KUKA KRL program: Kuka_Relative_Mo1.src

&ACCESS RVP
&REL 1
&PARAM TEMPLATE = C:\KRC\Roboter\Template\vorgabe
&PARAM EDITMASK = *
DEF Kuka_Relative_Mo1 ( )

; External program calls:
EXT Kuka_Relative_Mo2()

; $TOOL = TOOL_DATA[1]
; --------------------------
PTP {A1 -96.46360,A2 -64.41550,A3 114.80900,A4 -13.88510,A5 -54.29400,A6 -19.74150}
; ---- Setting reference (Base) ----
$BASE = {FRAME: X 0.000,Y 0.000,Z 0.000,A 0.000,B 0.000,C 0.000}
; --------------------------
; ---- Setting tool (TCP) ----
; TOOL_DATA[1] = {FRAME: X 0.000,Y 0.000,Z 10.000,A 0.000,B 0.000,C 0.000}
$TOOL = {FRAME: X 0.000,Y 0.000,Z 10.000,A 0.000,B 0.000,C 0.000}
; $TOOL = TOOL_DATA[1]
; --------------------------
PTP {A1 -96.46360,A2 -64.41550,A3 114.80900,A4 -13.88510,A5 -54.29400,A6 40.25850}
; ---- Setting reference (Base) ----
$BASE = {FRAME: X 0.000,Y 0.000,Z 0.000,A 0.000,B 0.000,C 0.000}
; --------------------------
; ---- Setting tool (TCP) ----
; TOOL_DATA[1] = {FRAME: X 0.000,Y 0.000,Z 10.000,A 0.000,B 0.000,C 0.000}
$TOOL = {FRAME: X 0.000,Y 0.000,Z 10.000,A 0.000,B 0.000,C 0.000}
; $TOOL = TOOL_DATA[1]
; --------------------------
PTP {A1 -96.46360,A2 -64.41550,A3 114.80900,A4 -13.88510,A5 -54.29400,A6 10.25850}
; ---- Setting reference (Base) ----
$BASE = {FRAME: X 0.000,Y 0.000,Z 0.000,A 0.000,B 0.000,C 0.000}
; --------------------------
; ---- Setting tool (TCP) ----
; TOOL_DATA[1] = {FRAME: X 0.000,Y 0.000,Z 10.000,A 0.000,B 0.000,C 0.000}
$TOOL = {FRAME: X 0.000,Y 0.000,Z 10.000,A 0.000,B 0.000,C 0.000}
; $TOOL = TOOL_DATA[1]
; --------------------------
PTP {A1 -85.55830,A2 -64.18770,A3 116.67500,A4 -0.42100,A5 -55.51980,A6 1.70277}
; ---- Setting reference (Base) ----
$BASE = {FRAME: X 0.000,Y 0.000,Z 0.000,A 0.000,B 0.000,C 0.000}
; --------------------------
; ---- Setting tool (TCP) ----
; TOOL_DATA[1] = {FRAME: X 0.000,Y 0.000,Z 10.000,A 0.000,B 0.000,C 0.000}
$TOOL = {FRAME: X 0.000,Y 0.000,Z 10.000,A 0.000,B 0.000,C 0.000}
; $TOOL = TOOL_DATA[1]
; --------------------------
PTP {A1 -90.55220,A2 -62.64360,A3 114.04900,A4 -40.68250,A5 -62.48120,A6 23.77200}
; ---- Setting reference (Base) ----
$BASE = {FRAME: X 0.000,Y 0.000,Z 0.000,A 0.000,B 0.000,C 0.000}
; --------------------------
; ---- Setting tool (TCP) ----
; TOOL_DATA[1] = {FRAME: X 0.000,Y 0.000,Z 10.000,A 0.000,B 0.000,C 0.000}
$TOOL = {FRAME: X 0.000,Y 0.000,Z 10.000,A 0.000,B 0.000,C 0.000}
; $TOOL = TOOL_DATA[1]
; --------------------------
PTP {A1 -80.54180,A2 -63.03590,A3 114.13400,A4 40.72610,A5 -60.63820,A6 -21.43390}
; ---- Setting reference (Base) ----
$BASE = {FRAME: X 0.000,Y 0.000,Z 0.000,A 0.000,B 0.000,C 0.000}
; --------------------------
; ---- Setting tool (TCP) ----
; TOOL_DATA[1] = {FRAME: X 0.000,Y 0.000,Z 10.000,A 0.000,B 0.000,C 0.000}
$TOOL = {FRAME: X 0.000,Y 0.000,Z 10.000,A 0.000,B 0.000,C 0.000}
; $TOOL = TOOL_DATA[1]
; --------------------------
PTP {A1 -85.55830,A2 -64.18770,A3 116.67500,A4 -0.42100,A5 -55.51980,A6 1.70277}
; ---- Setting reference (Base) ----
$BASE = {FRAME: X 0.000,Y 0.000,Z 0.000,A 0.000,B 0.000,C 0.000}
; --------------------------
; ---- Setting tool (TCP) ----
; TOOL_DATA[1] = {FRAME: X 0.000,Y 0.000,Z 10.000,A 0.000,B 0.000,C 0.000}
$TOOL = {FRAME: X 0.000,Y 0.000,Z 10.000,A 0.000,B 0.000,C 0.000}
; $TOOL = TOOL_DATA[1]
; --------------------------
PTP {A1 -85.55830,A2 -64.18770,A3 116.67500,A4 -0.42100,A5 -55.51980,A6 -28.29720}
; ---- Setting reference (Base) ----
$BASE = {FRAME: X 0.000,Y 0.000,Z 0.000,A 0.000,B 0.000,C 0.000}
; --------------------------
; ---- Setting tool (TCP) ----
; TOOL_DATA[1] = {FRAME: X 0.000,Y 0.000,Z 10.000,A 0.000,B 0.000,C 0.000}
$TOOL = {FRAME: X 0.000,Y 0.000,Z 10.000,A 0.000,B 0.000,C 0.000}
; $TOOL = TOOL_DATA[1]
; --------------------------
PTP {A1 -85.55830,A2 -64.18770,A3 116.67500,A4 -0.42100,A5 -55.51980,A6 31.70280}
; ---- Setting reference (Base) ----
$BASE = {FRAME: X 0.000,Y 0.000,Z 0.000,A 0.000,B 0.000,C 0.000}
; --------------------------
; ---- Setting tool (TCP) ----
; TOOL_DATA[1] = {FRAME: X 0.000,Y 0.000,Z 10.000,A 0.000,B 0.000,C 0.000}
$TOOL = {FRAME: X 0.000,Y 0.000,Z 10.000,A 0.000,B 0.000,C 0.000}
; $TOOL = TOOL_DATA[1]
; --------------------------
PTP {A1 -85.55830,A2 -64.18770,A3 116.67500,A4 -0.42100,A5 -55.51980,A6 1.70277}
; ---- Setting reference (Base) ----
$BASE = {FRAME: X 0.000,Y 0.000,Z 0.000,A 0.000,B 0.000,C 0.000}
; --------------------------
; ---- Setting tool (TCP) ----
; TOOL_DATA[1] = {FRAME: X 0.000,Y 0.000,Z 10.000,A 0.000,B 0.000,C 0.000}
$TOOL = {FRAME: X 0.000,Y 0.000,Z 10.000,A 0.000,B 0.000,C 0.000}
; $TOOL = TOOL_DATA[1]
; --------------------------
PTP {A1 -86.78140,A2 -64.12760,A3 116.64400,A4 -1.90174,A5 -55.56400,A6 2.60482}
; ---- Setting reference (Base) ----
$BASE = {FRAME: X 0.000,Y 0.000,Z 0.000,A 0.000,B 0.000,C 0.000}
; --------------------------
; ---- Setting tool (TCP) ----
; TOOL_DATA[1] = {FRAME: X 0.000,Y 0.000,Z 10.000,A 0.000,B 0.000,C 0.000}
$TOOL = {FRAME: X 0.000,Y 0.000,Z 10.000,A 0.000,B 0.000,C 0.000}
; $TOOL = TOOL_DATA[1]
; --------------------------
PTP {A1 -91.73390,A2 -62.48970,A3 113.84600,A4 -41.90860,A5 -62.93070,A6 24.43230}
; ---- Setting reference (Base) ----
$BASE = {FRAME: X 0.000,Y 0.000,Z 0.000,A 0.000,B 0.000,C 0.000}
; --------------------------
; ---- Setting tool (TCP) ----
; TOOL_DATA[1] = {FRAME: X 0.000,Y 0.000,Z 10.000,A 0.000,B 0.000,C 0.000}
$TOOL = {FRAME: X 0.000,Y 0.000,Z 10.000,A 0.000,B 0.000,C 0.000}
; $TOOL = TOOL_DATA[1]
; --------------------------
PTP {A1 -81.73080,A2 -63.07460,A3 114.27600,A4 39.43850,A5 -60.23740,A6 -20.70100}
; ---- Setting reference (Base) ----
$BASE = {FRAME: X 0.000,Y 0.000,Z 0.000,A 0.000,B 0.000,C 0.000}
; --------------------------
; ---- Setting tool (TCP) ----
; TOOL_DATA[1] = {FRAME: X 0.000,Y 0.000,Z 10.000,A 0.000,B 0.000,C 0.000}
$TOOL = {FRAME: X 0.000,Y 0.000,Z 10.000,A 0.000,B 0.000,C 0.000}
; $TOOL = TOOL_DATA[1]
; --------------------------
PTP {A1 -86.78140,A2 -64.12760,A3 116.64400,A4 -1.90174,A5 -55.56400,A6 2.60482}
; ---- Setting reference (Base) ----
$BASE = {FRAME: X 0.000,Y 0.000,Z 0.000,A 0.000,B 0.000,C 0.000}
; --------------------------
; ---- Setting tool (TCP) ----
; TOOL_DATA[1] = {FRAME: X 0.000,Y 0.000,Z 10.000,A 0.000,B 0.000,C 0.000}
$TOOL = {FRAME: X 0.000,Y 0.000,Z 10.000,A 0.000,B 0.000,C 0.000}
; $TOOL = TOOL_DATA[1]
; --------------------------
PTP {A1 -86.78140,A2 -64.12760,A3 116.64400,A4 -1.90174,A5 -55.56400,A6 -27.39520}
; ---- Setting reference (Base) ----
$BASE = {FRAME: X 0.000,Y 0.000,Z 0.000,A 0.000,B 0.000,C 0.000}
; --------------------------
; ---- Setting tool (TCP) ----
; TOOL_DATA[1] = {FRAME: X 0.000,Y 0.000,Z 10.000,A 0.000,B 0.000,C 0.000}
$TOOL = {FRAME: X 0.000,Y 0.000,Z 10.000,A 0.000,B 0.000,C 0.000}
; $TOOL = TOOL_DATA[1]
; --------------------------
PTP {A1 -86.78140,A2 -64.12760,A3 116.64400,A4 -1.90174,A5 -55.56400,A6 32.60480}
; ---- Setting reference (Base) ----
$BASE = {FRAME: X 0.000,Y 0.000,Z 0.000,A 0.000,B 0.000,C 0.000}
; --------------------------
; ---- Setting tool (TCP) ----
; TOOL_DATA[1] = {FRAME: X 0.000,Y 0.000,Z 10.000,A 0.000,B 0.000,C 0.000}
$TOOL = {FRAME: X 0.000,Y 0.000,Z 10.000,A 0.000,B 0.000,C 0.000}
; $TOOL = TOOL_DATA[1]
; --------------------------
PTP {A1 -86.78140,A2 -64.12760,A3 116.64400,A4 -1.90174,A5 -55.56400,A6 2.60482}
; ---- Setting reference (Base) ----
$BASE = {FRAME: X 0.000,Y 0.000,Z 0.000,A 0.000,B 0.000,C 0.000}
; --------------------------
; ---- Setting tool (TCP) ----
; TOOL_DATA[1] = {FRAME: X 0.000,Y 0.000,Z 10.000,A 0.000,B 0.000,C 0.000}
$TOOL = {FRAME: X 0.000,Y 0.000,Z 10.000,A 0.000,B 0.000,C 0.000}
; $TOOL = TOOL_DATA[1]
; --------------------------
PTP {A1 -88.00300,A2 -64.04420,A3 116.57100,A4 -3.37947,A5 -55.60900,A6 3.50421}
; ---- Setting reference (Base) ----
$BASE = {FRAME: X 0.000,Y 0.000,Z 0.000,A 0.000,B 0.000,C 0.000}
; --------------------------
; ---- Setting tool (TCP) ----
; TOOL_DATA[1] = {FRAME: X 0.000,Y 0.000,Z 10.000,A 0.000,B 0.000,C 0.000}
$TOOL = {FRAME: X 0.000,Y 0.000,Z 10.000,A 0.000,B 0.000,C 0.000}
; $TOOL = TOOL_DATA[1]
; --------------------------
PTP {A1 -92.91000,A2 -62.31340,A3 113.60200,A4 -43.12420,A5 -63.37720,A6 25.09110}
; ---- Setting reference (Base) ----
$BASE = {FRAME: X 0.000,Y 0.000,Z 0.000,A 0.000,B 0.000,C 0.000}
; --------------------------
; ---- Setting tool (TCP) ----
; TOOL_DATA[1] = {FRAME: X 0.000,Y 0.000,Z 10.000,A 0.000,B 0.000,C 0.000}
$TOOL = {FRAME: X 0.000,Y 0.000,Z 10.000,A 0.000,B 0.000,C 0.000}
; $TOOL = TOOL_DATA[1]
; --------------------------
PTP {A1 -82.92270,A2 -63.09010,A3 114.37700,A4 38.14280,A5 -59.83690,A6 -19.96770}
; ---- Setting reference (Base) ----
$BASE = {FRAME: X 0.000,Y 0.000,Z 0.000,A 0.000,B 0.000,C 0.000}
; --------------------------
; ---- Setting tool (TCP) ----
; TOOL_DATA[1] = {FRAME: X 0.000,Y 0.000,Z 10.000,A 0.000,B 0.000,C 0.000}
$TOOL = {FRAME: X 0.000,Y 0.000,Z 10.000,A 0.000,B 0.000,C 0.000}
; $TOOL = TOOL_DATA[1]
; --------------------------
PTP {A1 -88.00300,A2 -64.04420,A3 116.57100,A4 -3.37947,A5 -55.60900,A6 3.50421}
; ---- Setting reference (Base) ----
$BASE = {FRAME: X 0.000,Y 0.000,Z 0.000,A 0.000,B 0.000,C 0.000}
; --------------------------
; ---- Setting tool (TCP) ----
; TOOL_DATA[1] = {FRAME: X 0.000,Y 0.000,Z 10.000,A 0.000,B 0.000,C 0.000}
$TOOL = {FRAME: X 0.000,Y 0.000,Z 10.000,A 0.000,B 0.000,C 0.000}
; $TOOL = TOOL_DATA[1]
; --------------------------
PTP {A1 -88.00300,A2 -64.04420,A3 116.57100,A4 -3.37947,A5 -55.60900,A6 -26.49580}
; ---- Setting reference (Base) ----
$BASE = {FRAME: X 0.000,Y 0.000,Z 0.000,A 0.000,B 0.000,C 0.000}
; --------------------------
; ---- Setting tool (TCP) ----
; TOOL_DATA[1] = {FRAME: X 0.000,Y 0.000,Z 10.000,A 0.000,B 0.000,C 0.000}
$TOOL = {FRAME: X 0.000,Y 0.000,Z 10.000,A 0.000,B 0.000,C 0.000}
; $TOOL = TOOL_DATA[1]
; --------------------------
PTP {A1 -88.00300,A2 -64.04420,A3 116.57100,A4 -3.37947,A5 -55.60900,A6 33.50420}
; ---- Setting reference (Base) ----
$BASE = {FRAME: X 0.000,Y 0.000,Z 0.000,A 0.000,B 0.000,C 0.000}
; --------------------------
; ---- Setting tool (TCP) ----
; TOOL_DATA[1] = {FRAME: X 0.000,Y 0.000,Z 10.000,A 0.000,B 0.000,C 0.000}
$TOOL = {FRAME: X 0.000,Y 0.000,Z 10.000,A 0.000,B 0.000,C 0.000}
; $TOOL = TOOL_DATA[1]
; --------------------------
PTP {A1 -88.00300,A2 -64.04420,A3 116.57100,A4 -3.37947,A5 -55.60900,A6 3.50421}
; ---- Setting reference (Base) ----
$BASE = {FRAME: X 0.000,Y 0.000,Z 0.000,A 0.000,B 0.000,C 0.000}
; --------------------------
; ---- Setting tool (TCP) ----
; TOOL_DATA[1] = {FRAME: X 0.000,Y 0.000,Z 10.000,A 0.000,B 0.000,C 0.000}
$TOOL = {FRAME: X 0.000,Y 0.000,Z 10.000,A 0.000,B 0.000,C 0.000}
; $TOOL = TOOL_DATA[1]
; --------------------------
PTP {A1 -89.22190,A2 -63.93740,A3 116.45700,A4 -4.85314,A5 -55.65450,A6 4.40108}
; ---- Setting reference (Base) ----
$BASE = {FRAME: X 0.000,Y 0.000,Z 0.000,A 0.000,B 0.000,C 0.000}
; --------------------------
; ---- Setting tool (TCP) ----
; TOOL_DATA[1] = {FRAME: X 0.000,Y 0.000,Z 10.000,A 0.000,B 0.000,C 0.000}
$TOOL = {FRAME: X 0.000,Y 0.000,Z 10.000,A 0.000,B 0.000,C 0.000}
; $TOOL = TOOL_DATA[1]
; --------------------------
PTP {A1 -94.07950,A2 -62.11500,A3 113.31600,A4 -44.32860,A5 -63.82060,A6 25.74860}
; ---- Setting reference (Base) ----
$BASE = {FRAME: X 0.000,Y 0.000,Z 0.000,A 0.000,B 0.000,C 0.000}
; --------------------------
; ---- Setting tool (TCP) ----
; TOOL_DATA[1] = {FRAME: X 0.000,Y 0.000,Z 10.000,A 0.000,B 0.000,C 0.000}
$TOOL = {FRAME: X 0.000,Y 0.000,Z 10.000,A 0.000,B 0.000,C 0.000}
; $TOOL = TOOL_DATA[1]
; --------------------------
PTP {A1 -84.11650,A2 -63.08240,A3 114.43700,A4 36.83980,A5 -59.43650,A6 -19.23380}
; ---- Setting reference (Base) ----
$BASE = {FRAME: X 0.000,Y 0.000,Z 0.000,A 0.000,B 0.000,C 0.000}
; --------------------------
; ---- Setting tool (TCP) ----
; TOOL_DATA[1] = {FRAME: X 0.000,Y 0.000,Z 10.000,A 0.000,B 0.000,C 0.000}
$TOOL = {FRAME: X 0.000,Y 0.000,Z 10.000,A 0.000,B 0.000,C 0.000}
; $TOOL = TOOL_DATA[1]
; --------------------------
PTP {A1 -89.22190,A2 -63.93740,A3 116.45700,A4 -4.85314,A5 -55.65450,A6 4.40108}
; ---- Setting reference (Base) ----
$BASE = {FRAME: X 0.000,Y 0.000,Z 0.000,A 0.000,B 0.000,C 0.000}
; --------------------------
; ---- Setting tool (TCP) ----
; TOOL_DATA[1] = {FRAME: X 0.000,Y 0.000,Z 10.000,A 0.000,B 0.000,C 0.000}
$TOOL = {FRAME: X 0.000,Y 0.000,Z 10.000,A 0.000,B 0.000,C 0.000}
; $TOOL = TOOL_DATA[1]
; --------------------------
PTP {A1 -89.22190,A2 -63.93740,A3 116.45700,A4 -4.85314,A5 -55.65450,A6 -25.59890}
; ---- Setting reference (Base) ----
$BASE = {FRAME: X 0.000,Y 0.000,Z 0.000,A 0.000,B 0.000,C 0.000}
; --------------------------
; ---- Setting tool (TCP) ----
; TOOL_DATA[1] = {FRAME: X 0.000,Y 0.000,Z 10.000,A 0.000,B 0.000,C 0.000}
$TOOL = {FRAME: X 0.000,Y 0.000,Z 10.000,A 0.000,B 0.000,C 0.000}
; $TOOL = TOOL_DATA[1]
; --------------------------
PTP {A1 -89.22190,A2 -63.93740,A3 116.45700,A4 -4.85314,A5 -55.65450,A6 34.40110}
; ---- Setting reference (Base) ----
$BASE = {FRAME: X 0.000,Y 0.000,Z 0.000,A 0.000,B 0.000,C 0.000}
; --------------------------
; ---- Setting tool (TCP) ----
; TOOL_DATA[1] = {FRAME: X 0.000,Y 0.000,Z 10.000,A 0.000,B 0.000,C 0.000}
$TOOL = {FRAME: X 0.000,Y 0.000,Z 10.000,A 0.000,B 0.000,C 0.000}
; $TOOL = TOOL_DATA[1]
; --------------------------
PTP {A1 -89.22190,A2 -63.93740,A3 116.45700,A4 -4.85314,A5 -55.65450,A6 4.40108}
; ---- Setting reference (Base) ----
$BASE = {FRAME: X 0.000,Y 0.000,Z 0.000,A 0.000,B 0.000,C 0.000}
; --------------------------
; ---- Setting tool (TCP) ----
; TOOL_DATA[1] = {FRAME: X 0.000,Y 0.000,Z 10.000,A 0.000,B 0.000,C 0.000}
$TOOL = {FRAME: X 0.000,Y 0.000,Z 10.000,A 0.000,B 0.000,C 0.000}
; $TOOL = TOOL_DATA[1]
; --------------------------
PTP {A1 -90.43720,A2 -63.80760,A3 116.30100,A4 -6.32173,A5 -55.70030,A6 5.29557}
; ---- Setting reference (Base) ----
$BASE = {FRAME: X 0.000,Y 0.000,Z 0.000,A 0.000,B 0.000,C 0.000}
; --------------------------
; ---- Setting tool (TCP) ----
; TOOL_DATA[1] = {FRAME: X 0.000,Y 0.000,Z 10.000,A 0.000,B 0.000,C 0.000}
$TOOL = {FRAME: X 0.000,Y 0.000,Z 10.000,A 0.000,B 0.000,C 0.000}
; $TOOL = TOOL_DATA[1]
; --------------------------
PTP {A1 -95.24160,A2 -61.89470,A3 112.99100,A4 -45.52120,A5 -64.26070,A6 26.40550}
; ---- Setting reference (Base) ----
$BASE = {FRAME: X 0.000,Y 0.000,Z 0.000,A 0.000,B 0.000,C 0.000}
; --------------------------
; ---- Setting tool (TCP) ----
; TOOL_DATA[1] = {FRAME: X 0.000,Y 0.000,Z 10.000,A 0.000,B 0.000,C 0.000}
$TOOL = {FRAME: X 0.000,Y 0.000,Z 10.000,A 0.000,B 0.000,C 0.000}
; $TOOL = TOOL_DATA[1]
; --------------------------
PTP {A1 -85.31120,A2 -63.05160,A3 114.45600,A4 35.53070,A5 -59.03630,A6 -18.49930}
; ---- Setting reference (Base) ----
$BASE = {FRAME: X 0.000,Y 0.000,Z 0.000,A 0.000,B 0.000,C 0.000}
; --------------------------
; ---- Setting tool (TCP) ----
; TOOL_DATA[1] = {FRAME: X 0.000,Y 0.000,Z 10.000,A 0.000,B 0.000,C 0.000}
$TOOL = {FRAME: X 0.000,Y 0.000,Z 10.000,A 0.000,B 0.000,C 0.000}
; $TOOL = TOOL_DATA[1]
; --------------------------
PTP {A1 -90.43720,A2 -63.80760,A3 116.30100,A4 -6.32173,A5 -55.70030,A6 5.29557}
; ---- Setting reference (Base) ----
$BASE = {FRAME: X 0.000,Y 0.000,Z 0.000,A 0.000,B 0.000,C 0.000}
; --------------------------
; ---- Setting tool (TCP) ----
; TOOL_DATA[1] = {FRAME: X 0.000,Y 0.000,Z 10.000,A 0.000,B 0.000,C 0.000}
$TOOL = {FRAME: X 0.000,Y 0.000,Z 10.000,A 0.000,B 0.000,C 0.000}
; $TOOL = TOOL_DATA[1]
; --------------------------
PTP {A1 -90.43720,A2 -63.80760,A3 116.30100,A4 -6.32173,A5 -55.70030,A6 -24.70440}
; ---- Setting reference (Base) ----
$BASE = {FRAME: X 0.000,Y 0.000,Z 0.000,A 0.000,B 0.000,C 0.000}
; --------------------------
; ---- Setting tool (TCP) ----
; TOOL_DATA[1] = {FRAME: X 0.000,Y 0.000,Z 10.000,A 0.000,B 0.000,C 0.000}
$TOOL = {FRAME: X 0.000,Y 0.000,Z 10.000,A 0.000,B 0.000,C 0.000}
; $TOOL = TOOL_DATA[1]
; --------------------------
PTP {A1 -90.43720,A2 -63.80760,A3 116.30100,A4 -6.32173,A5 -55.70030,A6 35.29560}
; ---- Setting reference (Base) ----
$BASE = {FRAME: X 0.000,Y 0.000,Z 0.000,A 0.000,B 0.000,C 0.000}
; --------------------------
; ---- Setting tool (TCP) ----
; TOOL_DATA[1] = {FRAME: X 0.000,Y 0.000,Z 10.000,A 0.000,B 0.000,C 0.000}
$TOOL = {FRAME: X 0.000,Y 0.000,Z 10.000,A 0.000,B 0.000,C 0.000}
; $TOOL = TOOL_DATA[1]
; --------------------------
PTP {A1 -90.43720,A2 -63.80760,A3 116.30100,A4 -6.32173,A5 -55.70030,A6 5.29557}
; ---- Setting reference (Base) ----
$BASE = {FRAME: X 0.000,Y 0.000,Z 0.000,A 0.000,B 0.000,C 0.000}
; --------------------------
; ---- Setting tool (TCP) ----
; TOOL_DATA[1] = {FRAME: X 0.000,Y 0.000,Z 10.000,A 0.000,B 0.000,C 0.000}
$TOOL = {FRAME: X 0.000,Y 0.000,Z 10.000,A 0.000,B 0.000,C 0.000}
; $TOOL = TOOL_DATA[1]
; --------------------------
PTP {A1 -91.64770,A2 -63.65490,A3 116.10300,A4 -7.78425,A5 -55.74630,A6 6.18785}
; ---- Setting reference (Base) ----
$BASE = {FRAME: X 0.000,Y 0.000,Z 0.000,A 0.000,B 0.000,C 0.000}
; --------------------------
; ---- Setting tool (TCP) ----
; TOOL_DATA[1] = {FRAME: X 0.000,Y 0.000,Z 10.000,A 0.000,B 0.000,C 0.000}
$TOOL = {FRAME: X 0.000,Y 0.000,Z 10.000,A 0.000,B 0.000,C 0.000}
; $TOOL = TOOL_DATA[1]
; --------------------------
PTP {A1 -96.39530,A2 -61.65270,A3 112.62500,A4 -46.70110,A5 -64.69750,A6 27.06200}
; ---- Setting reference (Base) ----
$BASE = {FRAME: X 0.000,Y 0.000,Z 0.000,A 0.000,B 0.000,C 0.000}
; --------------------------
; ---- Setting tool (TCP) ----
; TOOL_DATA[1] = {FRAME: X 0.000,Y 0.000,Z 10.000,A 0.000,B 0.000,C 0.000}
$TOOL = {FRAME: X 0.000,Y 0.000,Z 10.000,A 0.000,B 0.000,C 0.000}
; $TOOL = TOOL_DATA[1]
; --------------------------
PTP {A1 -86.50580,A2 -62.99780,A3 114.43400,A4 34.21640,A5 -58.63620,A6 -17.76410}
; ---- Setting reference (Base) ----
$BASE = {FRAME: X 0.000,Y 0.000,Z 0.000,A 0.000,B 0.000,C 0.000}
; --------------------------
; ---- Setting tool (TCP) ----
; TOOL_DATA[1] = {FRAME: X 0.000,Y 0.000,Z 10.000,A 0.000,B 0.000,C 0.000}
$TOOL = {FRAME: X 0.000,Y 0.000,Z 10.000,A 0.000,B 0.000,C 0.000}
; $TOOL = TOOL_DATA[1]
; --------------------------
PTP {A1 -91.64770,A2 -63.65490,A3 116.10300,A4 -7.78425,A5 -55.74630,A6 6.18785}
; ---- Setting reference (Base) ----
$BASE = {FRAME: X 0.000,Y 0.000,Z 0.000,A 0.000,B 0.000,C 0.000}
; --------------------------
; ---- Setting tool (TCP) ----
; TOOL_DATA[1] = {FRAME: X 0.000,Y 0.000,Z 10.000,A 0.000,B 0.000,C 0.000}
$TOOL = {FRAME: X 0.000,Y 0.000,Z 10.000,A 0.000,B 0.000,C 0.000}
; $TOOL = TOOL_DATA[1]
; --------------------------
PTP {A1 -91.64770,A2 -63.65490,A3 116.10300,A4 -7.78425,A5 -55.74630,A6 -23.81210}
; ---- Setting reference (Base) ----
$BASE = {FRAME: X 0.000,Y 0.000,Z 0.000,A 0.000,B 0.000,C 0.000}
; --------------------------
; ---- Setting tool (TCP) ----
; TOOL_DATA[1] = {FRAME: X 0.000,Y 0.000,Z 10.000,A 0.000,B 0.000,C 0.000}
$TOOL = {FRAME: X 0.000,Y 0.000,Z 10.000,A 0.000,B 0.000,C 0.000}
; $TOOL = TOOL_DATA[1]
; --------------------------
PTP {A1 -91.64770,A2 -63.65490,A3 116.10300,A4 -7.78425,A5 -55.74630,A6 36.18790}
; ---- Setting reference (Base) ----
$BASE = {FRAME: X 0.000,Y 0.000,Z 0.000,A 0.000,B 0.000,C 0.000}
; --------------------------
; ---- Setting tool (TCP) ----
; TOOL_DATA[1] = {FRAME: X 0.000,Y 0.000,Z 10.000,A 0.000,B 0.000,C 0.000}
$TOOL = {FRAME: X 0.000,Y 0.000,Z 10.000,A 0.000,B 0.000,C 0.000}
; $TOOL = TOOL_DATA[1]
; --------------------------
PTP {A1 -91.64770,A2 -63.65490,A3 116.10300,A4 -7.78425,A5 -55.74630,A6 6.18785}
; ---- Setting reference (Base) ----
$BASE = {FRAME: X 0.000,Y 0.000,Z 0.000,A 0.000,B 0.000,C 0.000}
; --------------------------
; ---- Setting tool (TCP) ----
; TOOL_DATA[1] = {FRAME: X 0.000,Y 0.000,Z 10.000,A 0.000,B 0.000,C 0.000}
$TOOL = {FRAME: X 0.000,Y 0.000,Z 10.000,A 0.000,B 0.000,C 0.000}
; $TOOL = TOOL_DATA[1]
; --------------------------
PTP {A1 -92.85230,A2 -63.47960,A3 115.86400,A4 -9.23975,A5 -55.79220,A6 7.07814}
; ---- Setting reference (Base) ----
$BASE = {FRAME: X 0.000,Y 0.000,Z 0.000,A 0.000,B 0.000,C 0.000}
; --------------------------
; ---- Setting tool (TCP) ----
; TOOL_DATA[1] = {FRAME: X 0.000,Y 0.000,Z 10.000,A 0.000,B 0.000,C 0.000}
$TOOL = {FRAME: X 0.000,Y 0.000,Z 10.000,A 0.000,B 0.000,C 0.000}
; $TOOL = TOOL_DATA[1]
; --------------------------
PTP {A1 -97.53980,A2 -61.38930,A3 112.21800,A4 -47.86770,A5 -65.13090,A6 27.71860}
; ---- Setting reference (Base) ----
$BASE = {FRAME: X 0.000,Y 0.000,Z 0.000,A 0.000,B 0.000,C 0.000}
; --------------------------
; ---- Setting tool (TCP) ----
; TOOL_DATA[1] = {FRAME: X 0.000,Y 0.000,Z 10.000,A 0.000,B 0.000,C 0.000}
$TOOL = {FRAME: X 0.000,Y 0.000,Z 10.000,A 0.000,B 0.000,C 0.000}
; $TOOL = TOOL_DATA[1]
; --------------------------
PTP {A1 -87.69920,A2 -62.92100,A3 114.37000,A4 32.89790,A5 -58.23600,A6 -17.02810}
; ---- Setting reference (Base) ----
$BASE = {FRAME: X 0.000,Y 0.000,Z 0.000,A 0.000,B 0.000,C 0.000}
; --------------------------
; ---- Setting tool (TCP) ----
; TOOL_DATA[1] = {FRAME: X 0.000,Y 0.000,Z 10.000,A 0.000,B 0.000,C 0.000}
$TOOL = {FRAME: X 0.000,Y 0.000,Z 10.000,A 0.000,B 0.000,C 0.000}
; $TOOL = TOOL_DATA[1]
; --------------------------
PTP {A1 -92.85230,A2 -63.47960,A3 115.86400,A4 -9.23975,A5 -55.79220,A6 7.07814}
; ---- Setting reference (Base) ----
$BASE = {FRAME: X 0.000,Y 0.000,Z 0.000,A 0.000,B 0.000,C 0.000}
; --------------------------
; ---- Setting tool (TCP) ----
; TOOL_DATA[1] = {FRAME: X 0.000,Y 0.000,Z 10.000,A 0.000,B 0.000,C 0.000}
$TOOL = {FRAME: X 0.000,Y 0.000,Z 10.000,A 0.000,B 0.000,C 0.000}
; $TOOL = TOOL_DATA[1]
; --------------------------
PTP {A1 -92.85230,A2 -63.47960,A3 115.86400,A4 -9.23975,A5 -55.79220,A6 -22.92190}
; ---- Setting reference (Base) ----
$BASE = {FRAME: X 0.000,Y 0.000,Z 0.000,A 0.000,B 0.000,C 0.000}
; --------------------------
; ---- Setting tool (TCP) ----
; TOOL_DATA[1] = {FRAME: X 0.000,Y 0.000,Z 10.000,A 0.000,B 0.000,C 0.000}
$TOOL = {FRAME: X 0.000,Y 0.000,Z 10.000,A 0.000,B 0.000,C 0.000}
; $TOOL = TOOL_DATA[1]
; --------------------------
PTP {A1 -92.85230,A2 -63.47960,A3 115.86400,A4 -9.23975,A5 -55.79220,A6 37.07810}
; ---- Setting reference (Base) ----
$BASE = {FRAME: X 0.000,Y 0.000,Z 0.000,A 0.000,B 0.000,C 0.000}
; --------------------------
; ---- Setting tool (TCP) ----
; TOOL_DATA[1] = {FRAME: X 0.000,Y 0.000,Z 10.000,A 0.000,B 0.000,C 0.000}
$TOOL = {FRAME: X 0.000,Y 0.000,Z 10.000,A 0.000,B 0.000,C 0.000}
; $TOOL = TOOL_DATA[1]
; --------------------------
PTP {A1 -92.85230,A2 -63.47960,A3 115.86400,A4 -9.23975,A5 -55.79220,A6 7.07814}
; ---- Setting reference (Base) ----
$BASE = {FRAME: X 0.000,Y 0.000,Z 0.000,A 0.000,B 0.000,C 0.000}
; --------------------------
; ---- Setting tool (TCP) ----
; TOOL_DATA[1] = {FRAME: X 0.000,Y 0.000,Z 10.000,A 0.000,B 0.000,C 0.000}
$TOOL = {FRAME: X 0.000,Y 0.000,Z 10.000,A 0.000,B 0.000,C 0.000}
; $TOOL = TOOL_DATA[1]
; --------------------------
PTP {A1 -94.05020,A2 -63.28170,A3 115.58400,A4 -10.68730,A5 -55.83780,A6 7.96665}
; ---- Setting reference (Base) ----
$BASE = {FRAME: X 0.000,Y 0.000,Z 0.000,A 0.000,B 0.000,C 0.000}
; --------------------------
; ---- Setting tool (TCP) ----
; TOOL_DATA[1] = {FRAME: X 0.000,Y 0.000,Z 10.000,A 0.000,B 0.000,C 0.000}
$TOOL = {FRAME: X 0.000,Y 0.000,Z 10.000,A 0.000,B 0.000,C 0.000}
; $TOOL = TOOL_DATA[1]
; --------------------------
PTP {A1 -98.67440,A2 -61.10480,A3 111.77200,A4 -49.02040,A5 -65.56070,A6 28.37580}
; ---- Setting reference (Base) ----
$BASE = {FRAME: X 0.000,Y 0.000,Z 0.000,A 0.000,B 0.000,C 0.000}
; --------------------------
; ---- Setting tool (TCP) ----
; TOOL_DATA[1] = {FRAME: X 0.000,Y 0.000,Z 10.000,A 0.000,B 0.000,C 0.000}
$TOOL = {FRAME: X 0.000,Y 0.000,Z 10.000,A 0.000,B 0.000,C 0.000}
; $TOOL = TOOL_DATA[1]
; --------------------------
PTP {A1 -88.89030,A2 -62.82130,A3 114.26500,A4 31.57630,A5 -57.83560,A6 -16.29120}
; ---- Setting reference (Base) ----
$BASE = {FRAME: X 0.000,Y 0.000,Z 0.000,A 0.000,B 0.000,C 0.000}
; --------------------------
; ---- Setting tool (TCP) ----
; TOOL_DATA[1] = {FRAME: X 0.000,Y 0.000,Z 10.000,A 0.000,B 0.000,C 0.000}
$TOOL = {FRAME: X 0.000,Y 0.000,Z 10.000,A 0.000,B 0.000,C 0.000}
; $TOOL = TOOL_DATA[1]
; --------------------------
PTP {A1 -94.05020,A2 -63.28170,A3 115.58400,A4 -10.68730,A5 -55.83780,A6 7.96665}
; ---- Setting reference (Base) ----
$BASE = {FRAME: X 0.000,Y 0.000,Z 0.000,A 0.000,B 0.000,C 0.000}
; --------------------------
; ---- Setting tool (TCP) ----
; TOOL_DATA[1] = {FRAME: X 0.000,Y 0.000,Z 10.000,A 0.000,B 0.000,C 0.000}
$TOOL = {FRAME: X 0.000,Y 0.000,Z 10.000,A 0.000,B 0.000,C 0.000}
; $TOOL = TOOL_DATA[1]
; --------------------------
PTP {A1 -94.05020,A2 -63.28170,A3 115.58400,A4 -10.68730,A5 -55.83780,A6 -22.03340}
; ---- Setting reference (Base) ----
$BASE = {FRAME: X 0.000,Y 0.000,Z 0.000,A 0.000,B 0.000,C 0.000}
; --------------------------
; ---- Setting tool (TCP) ----
; TOOL_DATA[1] = {FRAME: X 0.000,Y 0.000,Z 10.000,A 0.000,B 0.000,C 0.000}
$TOOL = {FRAME: X 0.000,Y 0.000,Z 10.000,A 0.000,B 0.000,C 0.000}
; $TOOL = TOOL_DATA[1]
; --------------------------
PTP {A1 -94.05020,A2 -63.28170,A3 115.58400,A4 -10.68730,A5 -55.83780,A6 37.96660}
; ---- Setting reference (Base) ----
$BASE = {FRAME: X 0.000,Y 0.000,Z 0.000,A 0.000,B 0.000,C 0.000}
; --------------------------
; ---- Setting tool (TCP) ----
; TOOL_DATA[1] = {FRAME: X 0.000,Y 0.000,Z 10.000,A 0.000,B 0.000,C 0.000}
$TOOL = {FRAME: X 0.000,Y 0.000,Z 10.000,A 0.000,B 0.000,C 0.000}
; $TOOL = TOOL_DATA[1]
; --------------------------
PTP {A1 -94.05020,A2 -63.28170,A3 115.58400,A4 -10.68730,A5 -55.83780,A6 7.96665}
; ---- Setting reference (Base) ----
$BASE = {FRAME: X 0.000,Y 0.000,Z 0.000,A 0.000,B 0.000,C 0.000}
; --------------------------
; ---- Setting tool (TCP) ----
; TOOL_DATA[1] = {FRAME: X 0.000,Y 0.000,Z 10.000,A 0.000,B 0.000,C 0.000}
$TOOL = {FRAME: X 0.000,Y 0.000,Z 10.000,A 0.000,B 0.000,C 0.000}
; $TOOL = TOOL_DATA[1]
; --------------------------
PTP {A1 -95.24030,A2 -63.06160,A3 115.26300,A4 -12.12610,A5 -55.88270,A6 8.85365}
; ---- Setting reference (Base) ----
$BASE = {FRAME: X 0.000,Y 0.000,Z 0.000,A 0.000,B 0.000,C 0.000}
; --------------------------
; ---- Setting tool (TCP) ----
; TOOL_DATA[1] = {FRAME: X 0.000,Y 0.000,Z 10.000,A 0.000,B 0.000,C 0.000}
$TOOL = {FRAME: X 0.000,Y 0.000,Z 10.000,A 0.000,B 0.000,C 0.000}
; $TOOL = TOOL_DATA[1]
; --------------------------
PTP {A1 -99.79820,A2 -60.79930,A3 111.28600,A4 -50.15860,A5 -65.98710,A6 29.03400}
; ---- Setting reference (Base) ----
$BASE = {FRAME: X 0.000,Y 0.000,Z 0.000,A 0.000,B 0.000,C 0.000}
; --------------------------
; ---- Setting tool (TCP) ----
; TOOL_DATA[1] = {FRAME: X 0.000,Y 0.000,Z 10.000,A 0.000,B 0.000,C 0.000}
$TOOL = {FRAME: X 0.000,Y 0.000,Z 10.000,A 0.000,B 0.000,C 0.000}
; $TOOL = TOOL_DATA[1]
; --------------------------
PTP {A1 -90.07820,A2 -62.69890,A3 114.11900,A4 30.25250,A5 -57.43480,A6 -15.55340}
; ---- Setting reference (Base) ----
$BASE = {FRAME: X 0.000,Y 0.000,Z 0.000,A 0.000,B 0.000,C 0.000}
; --------------------------
; ---- Setting tool (TCP) ----
; TOOL_DATA[1] = {FRAME: X 0.000,Y 0.000,Z 10.000,A 0.000,B 0.000,C 0.000}
$TOOL = {FRAME: X 0.000,Y 0.000,Z 10.000,A 0.000,B 0.000,C 0.000}
; $TOOL = TOOL_DATA[1]
; --------------------------
PTP {A1 -95.24030,A2 -63.06160,A3 115.26300,A4 -12.12610,A5 -55.88270,A6 8.85365}
; ---- Setting reference (Base) ----
$BASE = {FRAME: X 0.000,Y 0.000,Z 0.000,A 0.000,B 0.000,C 0.000}
; --------------------------
; ---- Setting tool (TCP) ----
; TOOL_DATA[1] = {FRAME: X 0.000,Y 0.000,Z 10.000,A 0.000,B 0.000,C 0.000}
$TOOL = {FRAME: X 0.000,Y 0.000,Z 10.000,A 0.000,B 0.000,C 0.000}
; $TOOL = TOOL_DATA[1]
; --------------------------
PTP {A1 -95.24030,A2 -63.06160,A3 115.26300,A4 -12.12610,A5 -55.88270,A6 -21.14640}
; ---- Setting reference (Base) ----
$BASE = {FRAME: X 0.000,Y 0.000,Z 0.000,A 0.000,B 0.000,C 0.000}
; --------------------------
; ---- Setting tool (TCP) ----
; TOOL_DATA[1] = {FRAME: X 0.000,Y 0.000,Z 10.000,A 0.000,B 0.000,C 0.000}
$TOOL = {FRAME: X 0.000,Y 0.000,Z 10.000,A 0.000,B 0.000,C 0.000}
; $TOOL = TOOL_DATA[1]
; --------------------------
PTP {A1 -95.24030,A2 -63.06160,A3 115.26300,A4 -12.12610,A5 -55.88270,A6 38.85360}
; ---- Setting reference (Base) ----
$BASE = {FRAME: X 0.000,Y 0.000,Z 0.000,A 0.000,B 0.000,C 0.000}
; --------------------------
; ---- Setting tool (TCP) ----
; TOOL_DATA[1] = {FRAME: X 0.000,Y 0.000,Z 10.000,A 0.000,B 0.000,C 0.000}
$TOOL = {FRAME: X 0.000,Y 0.000,Z 10.000,A 0.000,B 0.000,C 0.000}
; $TOOL = TOOL_DATA[1]
; --------------------------
PTP {A1 -95.24030,A2 -63.06160,A3 115.26300,A4 -12.12610,A5 -55.88270,A6 8.85365}
; ---- Setting reference (Base) ----
$BASE = {FRAME: X 0.000,Y 0.000,Z 0.000,A 0.000,B 0.000,C 0.000}
; --------------------------
; ---- Setting tool (TCP) ----
; TOOL_DATA[1] = {FRAME: X 0.000,Y 0.000,Z 10.000,A 0.000,B 0.000,C 0.000}
$TOOL = {FRAME: X 0.000,Y 0.000,Z 10.000,A 0.000,B 0.000,C 0.000}
; $TOOL = TOOL_DATA[1]
; --------------------------
PTP {A1 -96.42160,A2 -62.81950,A3 114.90100,A4 -13.55530,A5 -55.92690,A6 9.73942}
; ---- Setting reference (Base) ----
$BASE = {FRAME: X 0.000,Y 0.000,Z 0.000,A 0.000,B 0.000,C 0.000}
; --------------------------
; ---- Setting tool (TCP) ----
; TOOL_DATA[1] = {FRAME: X 0.000,Y 0.000,Z 10.000,A 0.000,B 0.000,C 0.000}
$TOOL = {FRAME: X 0.000,Y 0.000,Z 10.000,A 0.000,B 0.000,C 0.000}
; $TOOL = TOOL_DATA[1]
; --------------------------
PTP {A1 -100.91100,A2 -60.47310,A3 110.76000,A4 -51.28180,A5 -66.40970,A6 29.69360}
; ---- Setting reference (Base) ----
$BASE = {FRAME: X 0.000,Y 0.000,Z 0.000,A 0.000,B 0.000,C 0.000}
; --------------------------
; ---- Setting tool (TCP) ----
; TOOL_DATA[1] = {FRAME: X 0.000,Y 0.000,Z 10.000,A 0.000,B 0.000,C 0.000}
$TOOL = {FRAME: X 0.000,Y 0.000,Z 10.000,A 0.000,B 0.000,C 0.000}
; $TOOL = TOOL_DATA[1]
; --------------------------
PTP {A1 -91.26190,A2 -62.55390,A3 113.93200,A4 28.92750,A5 -57.03360,A6 -14.81440}
; ---- Setting reference (Base) ----
$BASE = {FRAME: X 0.000,Y 0.000,Z 0.000,A 0.000,B 0.000,C 0.000}
; --------------------------
; ---- Setting tool (TCP) ----
; TOOL_DATA[1] = {FRAME: X 0.000,Y 0.000,Z 10.000,A 0.000,B 0.000,C 0.000}
$TOOL = {FRAME: X 0.000,Y 0.000,Z 10.000,A 0.000,B 0.000,C 0.000}
; $TOOL = TOOL_DATA[1]
; --------------------------
PTP {A1 -96.42160,A2 -62.81950,A3 114.90100,A4 -13.55530,A5 -55.92690,A6 9.73942}
; ---- Setting reference (Base) ----
$BASE = {FRAME: X 0.000,Y 0.000,Z 0.000,A 0.000,B 0.000,C 0.000}
; --------------------------
; ---- Setting tool (TCP) ----
; TOOL_DATA[1] = {FRAME: X 0.000,Y 0.000,Z 10.000,A 0.000,B 0.000,C 0.000}
$TOOL = {FRAME: X 0.000,Y 0.000,Z 10.000,A 0.000,B 0.000,C 0.000}
; $TOOL = TOOL_DATA[1]
; --------------------------
PTP {A1 -96.42160,A2 -62.81950,A3 114.90100,A4 -13.55530,A5 -55.92690,A6 -20.26060}
; ---- Setting reference (Base) ----
$BASE = {FRAME: X 0.000,Y 0.000,Z 0.000,A 0.000,B 0.000,C 0.000}
; --------------------------
; ---- Setting tool (TCP) ----
; TOOL_DATA[1] = {FRAME: X 0.000,Y 0.000,Z 10.000,A 0.000,B 0.000,C 0.000}
$TOOL = {FRAME: X 0.000,Y 0.000,Z 10.000,A 0.000,B 0.000,C 0.000}
; $TOOL = TOOL_DATA[1]
; --------------------------
PTP {A1 -96.42160,A2 -62.81950,A3 114.90100,A4 -13.55530,A5 -55.92690,A6 39.73940}
; ---- Setting reference (Base) ----
$BASE = {FRAME: X 0.000,Y 0.000,Z 0.000,A 0.000,B 0.000,C 0.000}
; --------------------------
; ---- Setting tool (TCP) ----
; TOOL_DATA[1] = {FRAME: X 0.000,Y 0.000,Z 10.000,A 0.000,B 0.000,C 0.000}
$TOOL = {FRAME: X 0.000,Y 0.000,Z 10.000,A 0.000,B 0.000,C 0.000}
; $TOOL = TOOL_DATA[1]
; --------------------------
PTP {A1 -96.42160,A2 -62.81950,A3 114.90100,A4 -13.55530,A5 -55.92690,A6 9.73942}
; ---- Setting reference (Base) ----
$BASE = {FRAME: X 0.000,Y 0.000,Z 0.000,A 0.000,B 0.000,C 0.000}
; --------------------------
; ---- Setting tool (TCP) ----
; TOOL_DATA[1] = {FRAME: X 0.000,Y 0.000,Z 10.000,A 0.000,B 0.000,C 0.000}
$TOOL = {FRAME: X 0.000,Y 0.000,Z 10.000,A 0.000,B 0.000,C 0.000}
; $TOOL = TOOL_DATA[1]
; --------------------------
PTP {A1 -85.52710,A2 -62.51940,A3 116.71400,A4 -0.37563,A5 -57.22740,A6 1.66612}
; ---- Setting reference (Base) ----
$BASE = {FRAME: X 0.000,Y 0.000,Z 0.000,A 0.000,B 0.000,C 0.000}
; --------------------------
; ---- Setting tool (TCP) ----
; TOOL_DATA[1] = {FRAME: X 0.000,Y 0.000,Z 10.000,A 0.000,B 0.000,C 0.000}
$TOOL = {FRAME: X 0.000,Y 0.000,Z 10.000,A 0.000,B 0.000,C 0.000}
; $TOOL = TOOL_DATA[1]
; --------------------------
PTP {A1 -90.51650,A2 -61.03770,A3 114.08600,A4 -40.10570,A5 -63.71800,A6 22.55980}
; ---- Setting reference (Base) ----
$BASE = {FRAME: X 0.000,Y 0.000,Z 0.000,A 0.000,B 0.000,C 0.000}
; --------------------------
; ---- Setting tool (TCP) ----
; TOOL_DATA[1] = {FRAME: X 0.000,Y 0.000,Z 10.000,A 0.000,B 0.000,C 0.000}
$TOOL = {FRAME: X 0.000,Y 0.000,Z 10.000,A 0.000,B 0.000,C 0.000}
; $TOOL = TOOL_DATA[1]
; --------------------------
PTP {A1 -80.51700,A2 -61.42930,A3 114.17400,A4 40.16640,A5 -61.90130,A6 -20.22910}
; ---- Setting reference (Base) ----
$BASE = {FRAME: X 0.000,Y 0.000,Z 0.000,A 0.000,B 0.000,C 0.000}
; --------------------------
; ---- Setting tool (TCP) ----
; TOOL_DATA[1] = {FRAME: X 0.000,Y 0.000,Z 10.000,A 0.000,B 0.000,C 0.000}
$TOOL = {FRAME: X 0.000,Y 0.000,Z 10.000,A 0.000,B 0.000,C 0.000}
; $TOOL = TOOL_DATA[1]
; --------------------------
PTP {A1 -85.52710,A2 -62.51940,A3 116.71400,A4 -0.37563,A5 -57.22740,A6 1.66612}
; ---- Setting reference (Base) ----
$BASE = {FRAME: X 0.000,Y 0.000,Z 0.000,A 0.000,B 0.000,C 0.000}
; --------------------------
; ---- Setting tool (TCP) ----
; TOOL_DATA[1] = {FRAME: X 0.000,Y 0.000,Z 10.000,A 0.000,B 0.000,C 0.000}
$TOOL = {FRAME: X 0.000,Y 0.000,Z 10.000,A 0.000,B 0.000,C 0.000}
; $TOOL = TOOL_DATA[1]
; --------------------------
PTP {A1 -85.52710,A2 -62.51940,A3 116.71400,A4 -0.37563,A5 -57.22740,A6 -28.33390}
; ---- Setting reference (Base) ----
$BASE = {FRAME: X 0.000,Y 0.000,Z 0.000,A 0.000,B 0.000,C 0.000}
; --------------------------
; ---- Setting tool (TCP) ----
; TOOL_DATA[1] = {FRAME: X 0.000,Y 0.000,Z 10.000,A 0.000,B 0.000,C 0.000}
$TOOL = {FRAME: X 0.000,Y 0.000,Z 10.000,A 0.000,B 0.000,C 0.000}
; $TOOL = TOOL_DATA[1]
; --------------------------
PTP {A1 -85.52710,A2 -62.51940,A3 116.71400,A4 -0.37563,A5 -57.22740,A6 31.66610}
; ---- Setting reference (Base) ----
$BASE = {FRAME: X 0.000,Y 0.000,Z 0.000,A 0.000,B 0.000,C 0.000}
; --------------------------
; ---- Setting tool (TCP) ----
; TOOL_DATA[1] = {FRAME: X 0.000,Y 0.000,Z 10.000,A 0.000,B 0.000,C 0.000}
$TOOL = {FRAME: X 0.000,Y 0.000,Z 10.000,A 0.000,B 0.000,C 0.000}
; $TOOL = TOOL_DATA[1]
; --------------------------
PTP {A1 -85.52710,A2 -62.51940,A3 116.71400,A4 -0.37563,A5 -57.22740,A6 1.66612}
; ---- Setting reference (Base) ----
$BASE = {FRAME: X 0.000,Y 0.000,Z 0.000,A 0.000,B 0.000,C 0.000}
; --------------------------
; ---- Setting tool (TCP) ----
; TOOL_DATA[1] = {FRAME: X 0.000,Y 0.000,Z 10.000,A 0.000,B 0.000,C 0.000}
$TOOL = {FRAME: X 0.000,Y 0.000,Z 10.000,A 0.000,B 0.000,C 0.000}
; $TOOL = TOOL_DATA[1]
; --------------------------
PTP {A1 -86.74880,A2 -62.45990,A3 116.68300,A4 -1.82581,A5 -57.26920,A6 2.51486}
; ---- Setting reference (Base) ----
$BASE = {FRAME: X 0.000,Y 0.000,Z 0.000,A 0.000,B 0.000,C 0.000}
; --------------------------
; ---- Setting tool (TCP) ----
; TOOL_DATA[1] = {FRAME: X 0.000,Y 0.000,Z 10.000,A 0.000,B 0.000,C 0.000}
$TOOL = {FRAME: X 0.000,Y 0.000,Z 10.000,A 0.000,B 0.000,C 0.000}
; $TOOL = TOOL_DATA[1]
; --------------------------
PTP {A1 -91.69710,A2 -60.88830,A3 113.88200,A4 -41.32960,A5 -64.13990,A6 23.19850}
; ---- Setting reference (Base) ----
$BASE = {FRAME: X 0.000,Y 0.000,Z 0.000,A 0.000,B 0.000,C 0.000}
; --------------------------
; ---- Setting tool (TCP) ----
; TOOL_DATA[1] = {FRAME: X 0.000,Y 0.000,Z 10.000,A 0.000,B 0.000,C 0.000}
$TOOL = {FRAME: X 0.000,Y 0.000,Z 10.000,A 0.000,B 0.000,C 0.000}
; $TOOL = TOOL_DATA[1]
; --------------------------
PTP {A1 -81.70460,A2 -61.46460,A3 114.31600,A4 38.88580,A5 -61.52670,A6 -19.52280}
; ---- Setting reference (Base) ----
$BASE = {FRAME: X 0.000,Y 0.000,Z 0.000,A 0.000,B 0.000,C 0.000}
; --------------------------
; ---- Setting tool (TCP) ----
; TOOL_DATA[1] = {FRAME: X 0.000,Y 0.000,Z 10.000,A 0.000,B 0.000,C 0.000}
$TOOL = {FRAME: X 0.000,Y 0.000,Z 10.000,A 0.000,B 0.000,C 0.000}
; $TOOL = TOOL_DATA[1]
; --------------------------
PTP {A1 -86.74880,A2 -62.45990,A3 116.68300,A4 -1.82581,A5 -57.26920,A6 2.51486}
; ---- Setting reference (Base) ----
$BASE = {FRAME: X 0.000,Y 0.000,Z 0.000,A 0.000,B 0.000,C 0.000}
; --------------------------
; ---- Setting tool (TCP) ----
; TOOL_DATA[1] = {FRAME: X 0.000,Y 0.000,Z 10.000,A 0.000,B 0.000,C 0.000}
$TOOL = {FRAME: X 0.000,Y 0.000,Z 10.000,A 0.000,B 0.000,C 0.000}
; $TOOL = TOOL_DATA[1]
; --------------------------
PTP {A1 -86.74880,A2 -62.45990,A3 116.68300,A4 -1.82581,A5 -57.26920,A6 -27.48510}
; ---- Setting reference (Base) ----
$BASE = {FRAME: X 0.000,Y 0.000,Z 0.000,A 0.000,B 0.000,C 0.000}
; --------------------------
; ---- Setting tool (TCP) ----
; TOOL_DATA[1] = {FRAME: X 0.000,Y 0.000,Z 10.000,A 0.000,B 0.000,C 0.000}
$TOOL = {FRAME: X 0.000,Y 0.000,Z 10.000,A 0.000,B 0.000,C 0.000}
; $TOOL = TOOL_DATA[1]
; --------------------------
PTP {A1 -86.74880,A2 -62.45990,A3 116.68300,A4 -1.82581,A5 -57.26920,A6 32.51490}
; ---- Setting reference (Base) ----
$BASE = {FRAME: X 0.000,Y 0.000,Z 0.000,A 0.000,B 0.000,C 0.000}
; --------------------------
; ---- Setting tool (TCP) ----
; TOOL_DATA[1] = {FRAME: X 0.000,Y 0.000,Z 10.000,A 0.000,B 0.000,C 0.000}
$TOOL = {FRAME: X 0.000,Y 0.000,Z 10.000,A 0.000,B 0.000,C 0.000}
; $TOOL = TOOL_DATA[1]
; --------------------------
PTP {A1 -86.74880,A2 -62.45990,A3 116.68300,A4 -1.82581,A5 -57.26920,A6 2.51486}
; ---- Setting reference (Base) ----
$BASE = {FRAME: X 0.000,Y 0.000,Z 0.000,A 0.000,B 0.000,C 0.000}
; --------------------------
; ---- Setting tool (TCP) ----
; TOOL_DATA[1] = {FRAME: X 0.000,Y 0.000,Z 10.000,A 0.000,B 0.000,C 0.000}
$TOOL = {FRAME: X 0.000,Y 0.000,Z 10.000,A 0.000,B 0.000,C 0.000}
; $TOOL = TOOL_DATA[1]
; --------------------------
PTP {A1 -87.96900,A2 -62.37810,A3 116.61000,A4 -3.27328,A5 -57.30950,A6 3.36131}
; ---- Setting reference (Base) ----
$BASE = {FRAME: X 0.000,Y 0.000,Z 0.000,A 0.000,B 0.000,C 0.000}
; --------------------------
; ---- Setting tool (TCP) ----
; TOOL_DATA[1] = {FRAME: X 0.000,Y 0.000,Z 10.000,A 0.000,B 0.000,C 0.000}
$TOOL = {FRAME: X 0.000,Y 0.000,Z 10.000,A 0.000,B 0.000,C 0.000}
; $TOOL = TOOL_DATA[1]
; --------------------------
PTP {A1 -92.87200,A2 -60.71740,A3 113.63700,A4 -42.54400,A5 -64.55790,A6 23.83750}
; ---- Setting reference (Base) ----
$BASE = {FRAME: X 0.000,Y 0.000,Z 0.000,A 0.000,B 0.000,C 0.000}
; --------------------------
; ---- Setting tool (TCP) ----
; TOOL_DATA[1] = {FRAME: X 0.000,Y 0.000,Z 10.000,A 0.000,B 0.000,C 0.000}
$TOOL = {FRAME: X 0.000,Y 0.000,Z 10.000,A 0.000,B 0.000,C 0.000}
; $TOOL = TOOL_DATA[1]
; --------------------------
PTP {A1 -82.89510,A2 -61.47760,A3 114.41700,A4 37.59820,A5 -61.15130,A6 -18.81790}
; ---- Setting reference (Base) ----
$BASE = {FRAME: X 0.000,Y 0.000,Z 0.000,A 0.000,B 0.000,C 0.000}
; --------------------------
; ---- Setting tool (TCP) ----
; TOOL_DATA[1] = {FRAME: X 0.000,Y 0.000,Z 10.000,A 0.000,B 0.000,C 0.000}
$TOOL = {FRAME: X 0.000,Y 0.000,Z 10.000,A 0.000,B 0.000,C 0.000}
; $TOOL = TOOL_DATA[1]
; --------------------------
PTP {A1 -87.96900,A2 -62.37810,A3 116.61000,A4 -3.27328,A5 -57.30950,A6 3.36131}
; ---- Setting reference (Base) ----
$BASE = {FRAME: X 0.000,Y 0.000,Z 0.000,A 0.000,B 0.000,C 0.000}
; --------------------------
; ---- Setting tool (TCP) ----
; TOOL_DATA[1] = {FRAME: X 0.000,Y 0.000,Z 10.000,A 0.000,B 0.000,C 0.000}
$TOOL = {FRAME: X 0.000,Y 0.000,Z 10.000,A 0.000,B 0.000,C 0.000}
; $TOOL = TOOL_DATA[1]
; --------------------------
PTP {A1 -87.96900,A2 -62.37810,A3 116.61000,A4 -3.27328,A5 -57.30950,A6 -26.63870}
; ---- Setting reference (Base) ----
$BASE = {FRAME: X 0.000,Y 0.000,Z 0.000,A 0.000,B 0.000,C 0.000}
; --------------------------
; ---- Setting tool (TCP) ----
; TOOL_DATA[1] = {FRAME: X 0.000,Y 0.000,Z 10.000,A 0.000,B 0.000,C 0.000}
$TOOL = {FRAME: X 0.000,Y 0.000,Z 10.000,A 0.000,B 0.000,C 0.000}
; $TOOL = TOOL_DATA[1]
; --------------------------
PTP {A1 -87.96900,A2 -62.37810,A3 116.61000,A4 -3.27328,A5 -57.30950,A6 33.36130}
; ---- Setting reference (Base) ----
$BASE = {FRAME: X 0.000,Y 0.000,Z 0.000,A 0.000,B 0.000,C 0.000}
; --------------------------
; ---- Setting tool (TCP) ----
; TOOL_DATA[1] = {FRAME: X 0.000,Y 0.000,Z 10.000,A 0.000,B 0.000,C 0.000}
$TOOL = {FRAME: X 0.000,Y 0.000,Z 10.000,A 0.000,B 0.000,C 0.000}
; $TOOL = TOOL_DATA[1]
; --------------------------
PTP {A1 -87.96900,A2 -62.37810,A3 116.61000,A4 -3.27328,A5 -57.30950,A6 3.36131}
; ---- Setting reference (Base) ----
$BASE = {FRAME: X 0.000,Y 0.000,Z 0.000,A 0.000,B 0.000,C 0.000}
; --------------------------
; ---- Setting tool (TCP) ----
; TOOL_DATA[1] = {FRAME: X 0.000,Y 0.000,Z 10.000,A 0.000,B 0.000,C 0.000}
$TOOL = {FRAME: X 0.000,Y 0.000,Z 10.000,A 0.000,B 0.000,C 0.000}
; $TOOL = TOOL_DATA[1]
; --------------------------
PTP {A1 -89.18670,A2 -62.27410,A3 116.49500,A4 -4.71709,A5 -57.34820,A6 4.20578}
; ---- Setting reference (Base) ----
$BASE = {FRAME: X 0.000,Y 0.000,Z 0.000,A 0.000,B 0.000,C 0.000}
; --------------------------
; ---- Setting tool (TCP) ----
; TOOL_DATA[1] = {FRAME: X 0.000,Y 0.000,Z 10.000,A 0.000,B 0.000,C 0.000}
$TOOL = {FRAME: X 0.000,Y 0.000,Z 10.000,A 0.000,B 0.000,C 0.000}
; $TOOL = TOOL_DATA[1]
; --------------------------
PTP {A1 -94.04050,A2 -60.52520,A3 113.35100,A4 -43.74830,A5 -64.97190,A6 24.47710}
; ---- Setting reference (Base) ----
$BASE = {FRAME: X 0.000,Y 0.000,Z 0.000,A 0.000,B 0.000,C 0.000}
; --------------------------
; ---- Setting tool (TCP) ----
; TOOL_DATA[1] = {FRAME: X 0.000,Y 0.000,Z 10.000,A 0.000,B 0.000,C 0.000}
$TOOL = {FRAME: X 0.000,Y 0.000,Z 10.000,A 0.000,B 0.000,C 0.000}
; $TOOL = TOOL_DATA[1]
; --------------------------
PTP {A1 -84.08760,A2 -61.46840,A3 114.47600,A4 36.30460,A5 -60.77470,A6 -18.11420}
; ---- Setting reference (Base) ----
$BASE = {FRAME: X 0.000,Y 0.000,Z 0.000,A 0.000,B 0.000,C 0.000}
; --------------------------
; ---- Setting tool (TCP) ----
; TOOL_DATA[1] = {FRAME: X 0.000,Y 0.000,Z 10.000,A 0.000,B 0.000,C 0.000}
$TOOL = {FRAME: X 0.000,Y 0.000,Z 10.000,A 0.000,B 0.000,C 0.000}
; $TOOL = TOOL_DATA[1]
; --------------------------
PTP {A1 -89.18670,A2 -62.27410,A3 116.49500,A4 -4.71709,A5 -57.34820,A6 4.20578}
; ---- Setting reference (Base) ----
$BASE = {FRAME: X 0.000,Y 0.000,Z 0.000,A 0.000,B 0.000,C 0.000}
; --------------------------
; ---- Setting tool (TCP) ----
; TOOL_DATA[1] = {FRAME: X 0.000,Y 0.000,Z 10.000,A 0.000,B 0.000,C 0.000}
$TOOL = {FRAME: X 0.000,Y 0.000,Z 10.000,A 0.000,B 0.000,C 0.000}
; $TOOL = TOOL_DATA[1]
; --------------------------
PTP {A1 -89.18670,A2 -62.27410,A3 116.49500,A4 -4.71709,A5 -57.34820,A6 -25.79420}
; ---- Setting reference (Base) ----
$BASE = {FRAME: X 0.000,Y 0.000,Z 0.000,A 0.000,B 0.000,C 0.000}
; --------------------------
; ---- Setting tool (TCP) ----
; TOOL_DATA[1] = {FRAME: X 0.000,Y 0.000,Z 10.000,A 0.000,B 0.000,C 0.000}
$TOOL = {FRAME: X 0.000,Y 0.000,Z 10.000,A 0.000,B 0.000,C 0.000}
; $TOOL = TOOL_DATA[1]
; --------------------------
PTP {A1 -89.18670,A2 -62.27410,A3 116.49500,A4 -4.71709,A5 -57.34820,A6 34.20580}
; ---- Setting reference (Base) ----
$BASE = {FRAME: X 0.000,Y 0.000,Z 0.000,A 0.000,B 0.000,C 0.000}
; --------------------------
; ---- Setting tool (TCP) ----
; TOOL_DATA[1] = {FRAME: X 0.000,Y 0.000,Z 10.000,A 0.000,B 0.000,C 0.000}
$TOOL = {FRAME: X 0.000,Y 0.000,Z 10.000,A 0.000,B 0.000,C 0.000}
; $TOOL = TOOL_DATA[1]
; --------------------------
PTP {A1 -89.18670,A2 -62.27410,A3 116.49500,A4 -4.71709,A5 -57.34820,A6 4.20578}
; ---- Setting reference (Base) ----
$BASE = {FRAME: X 0.000,Y 0.000,Z 0.000,A 0.000,B 0.000,C 0.000}
; --------------------------
; ---- Setting tool (TCP) ----
; TOOL_DATA[1] = {FRAME: X 0.000,Y 0.000,Z 10.000,A 0.000,B 0.000,C 0.000}
$TOOL = {FRAME: X 0.000,Y 0.000,Z 10.000,A 0.000,B 0.000,C 0.000}
; $TOOL = TOOL_DATA[1]
; --------------------------
PTP {A1 -90.40070,A2 -62.14800,A3 116.33800,A4 -6.15629,A5 -57.38510,A6 5.04857}
; ---- Setting reference (Base) ----
$BASE = {FRAME: X 0.000,Y 0.000,Z 0.000,A 0.000,B 0.000,C 0.000}
; --------------------------
; ---- Setting tool (TCP) ----
; TOOL_DATA[1] = {FRAME: X 0.000,Y 0.000,Z 10.000,A 0.000,B 0.000,C 0.000}
$TOOL = {FRAME: X 0.000,Y 0.000,Z 10.000,A 0.000,B 0.000,C 0.000}
; $TOOL = TOOL_DATA[1]
; --------------------------
PTP {A1 -95.20150,A2 -60.31200,A3 113.02500,A4 -44.94170,A5 -65.38210,A6 25.11770}
; ---- Setting reference (Base) ----
$BASE = {FRAME: X 0.000,Y 0.000,Z 0.000,A 0.000,B 0.000,C 0.000}
; --------------------------
; ---- Setting tool (TCP) ----
; TOOL_DATA[1] = {FRAME: X 0.000,Y 0.000,Z 10.000,A 0.000,B 0.000,C 0.000}
$TOOL = {FRAME: X 0.000,Y 0.000,Z 10.000,A 0.000,B 0.000,C 0.000}
; $TOOL = TOOL_DATA[1]
; --------------------------
PTP {A1 -85.28100,A2 -61.43700,A3 114.49500,A4 35.00590,A5 -60.39690,A6 -17.41140}
; ---- Setting reference (Base) ----
$BASE = {FRAME: X 0.000,Y 0.000,Z 0.000,A 0.000,B 0.000,C 0.000}
; --------------------------
; ---- Setting tool (TCP) ----
; TOOL_DATA[1] = {FRAME: X 0.000,Y 0.000,Z 10.000,A 0.000,B 0.000,C 0.000}
$TOOL = {FRAME: X 0.000,Y 0.000,Z 10.000,A 0.000,B 0.000,C 0.000}
; $TOOL = TOOL_DATA[1]
; --------------------------
PTP {A1 -90.40070,A2 -62.14800,A3 116.33800,A4 -6.15629,A5 -57.38510,A6 5.04857}
; ---- Setting reference (Base) ----
$BASE = {FRAME: X 0.000,Y 0.000,Z 0.000,A 0.000,B 0.000,C 0.000}
; --------------------------
; ---- Setting tool (TCP) ----
; TOOL_DATA[1] = {FRAME: X 0.000,Y 0.000,Z 10.000,A 0.000,B 0.000,C 0.000}
$TOOL = {FRAME: X 0.000,Y 0.000,Z 10.000,A 0.000,B 0.000,C 0.000}
; $TOOL = TOOL_DATA[1]
; --------------------------
PTP {A1 -90.40070,A2 -62.14800,A3 116.33800,A4 -6.15629,A5 -57.38510,A6 -24.95140}
; ---- Setting reference (Base) ----
$BASE = {FRAME: X 0.000,Y 0.000,Z 0.000,A 0.000,B 0.000,C 0.000}
; --------------------------
; ---- Setting tool (TCP) ----
; TOOL_DATA[1] = {FRAME: X 0.000,Y 0.000,Z 10.000,A 0.000,B 0.000,C 0.000}
$TOOL = {FRAME: X 0.000,Y 0.000,Z 10.000,A 0.000,B 0.000,C 0.000}
; $TOOL = TOOL_DATA[1]
; --------------------------
PTP {A1 -90.40070,A2 -62.14800,A3 116.33800,A4 -6.15629,A5 -57.38510,A6 35.04860}
; ---- Setting reference (Base) ----
$BASE = {FRAME: X 0.000,Y 0.000,Z 0.000,A 0.000,B 0.000,C 0.000}
; --------------------------
; ---- Setting tool (TCP) ----
; TOOL_DATA[1] = {FRAME: X 0.000,Y 0.000,Z 10.000,A 0.000,B 0.000,C 0.000}
$TOOL = {FRAME: X 0.000,Y 0.000,Z 10.000,A 0.000,B 0.000,C 0.000}
; $TOOL = TOOL_DATA[1]
; --------------------------
PTP {A1 -90.40070,A2 -62.14800,A3 116.33800,A4 -6.15629,A5 -57.38510,A6 5.04857}
; ---- Setting reference (Base) ----
$BASE = {FRAME: X 0.000,Y 0.000,Z 0.000,A 0.000,B 0.000,C 0.000}
; --------------------------
; ---- Setting tool (TCP) ----
; TOOL_DATA[1] = {FRAME: X 0.000,Y 0.000,Z 10.000,A 0.000,B 0.000,C 0.000}
$TOOL = {FRAME: X 0.000,Y 0.000,Z 10.000,A 0.000,B 0.000,C 0.000}
; $TOOL = TOOL_DATA[1]
; --------------------------
PTP {A1 -91.61000,A2 -62.00000,A3 116.14000,A4 -7.59000,A5 -57.42000,A6 5.89000}
; ---- Setting reference (Base) ----
$BASE = {FRAME: X 0.000,Y 0.000,Z 0.000,A 0.000,B 0.000,C 0.000}
; --------------------------
; ---- Setting tool (TCP) ----
; TOOL_DATA[1] = {FRAME: X 0.000,Y 0.000,Z 10.000,A 0.000,B 0.000,C 0.000}
$TOOL = {FRAME: X 0.000,Y 0.000,Z 10.000,A 0.000,B 0.000,C 0.000}
; $TOOL = TOOL_DATA[1]
; --------------------------
PTP {A1 -96.35430,A2 -60.07790,A3 112.65800,A4 -46.12340,A5 -65.78830,A6 25.75970}
; ---- Setting reference (Base) ----
$BASE = {FRAME: X 0.000,Y 0.000,Z 0.000,A 0.000,B 0.000,C 0.000}
; --------------------------
; ---- Setting tool (TCP) ----
; TOOL_DATA[1] = {FRAME: X 0.000,Y 0.000,Z 10.000,A 0.000,B 0.000,C 0.000}
$TOOL = {FRAME: X 0.000,Y 0.000,Z 10.000,A 0.000,B 0.000,C 0.000}
; $TOOL = TOOL_DATA[1]
; --------------------------
PTP {A1 -86.47430,A2 -61.38360,A3 114.47200,A4 33.70330,A5 -60.01760,A6 -16.70950}
; ---- Setting reference (Base) ----
$BASE = {FRAME: X 0.000,Y 0.000,Z 0.000,A 0.000,B 0.000,C 0.000}
; --------------------------
; ---- Setting tool (TCP) ----
; TOOL_DATA[1] = {FRAME: X 0.000,Y 0.000,Z 10.000,A 0.000,B 0.000,C 0.000}
$TOOL = {FRAME: X 0.000,Y 0.000,Z 10.000,A 0.000,B 0.000,C 0.000}
; $TOOL = TOOL_DATA[1]
; --------------------------
PTP {A1 -91.61000,A2 -62.00000,A3 116.14000,A4 -7.59000,A5 -57.42000,A6 5.89000}
; ---- Setting reference (Base) ----
$BASE = {FRAME: X 0.000,Y 0.000,Z 0.000,A 0.000,B 0.000,C 0.000}
; --------------------------
; ---- Setting tool (TCP) ----
; TOOL_DATA[1] = {FRAME: X 0.000,Y 0.000,Z 10.000,A 0.000,B 0.000,C 0.000}
$TOOL = {FRAME: X 0.000,Y 0.000,Z 10.000,A 0.000,B 0.000,C 0.000}
; $TOOL = TOOL_DATA[1]
; --------------------------
PTP {A1 -91.61000,A2 -62.00000,A3 116.14000,A4 -7.59000,A5 -57.42000,A6 -24.11000}
; ---- Setting reference (Base) ----
$BASE = {FRAME: X 0.000,Y 0.000,Z 0.000,A 0.000,B 0.000,C 0.000}
; --------------------------
; ---- Setting tool (TCP) ----
; TOOL_DATA[1] = {FRAME: X 0.000,Y 0.000,Z 10.000,A 0.000,B 0.000,C 0.000}
$TOOL = {FRAME: X 0.000,Y 0.000,Z 10.000,A 0.000,B 0.000,C 0.000}
; $TOOL = TOOL_DATA[1]
; --------------------------
PTP {A1 -91.61000,A2 -62.00000,A3 116.14000,A4 -7.59000,A5 -57.42000,A6 35.89000}
; ---- Setting reference (Base) ----
$BASE = {FRAME: X 0.000,Y 0.000,Z 0.000,A 0.000,B 0.000,C 0.000}
; --------------------------
; ---- Setting tool (TCP) ----
; TOOL_DATA[1] = {FRAME: X 0.000,Y 0.000,Z 10.000,A 0.000,B 0.000,C 0.000}
$TOOL = {FRAME: X 0.000,Y 0.000,Z 10.000,A 0.000,B 0.000,C 0.000}
; $TOOL = TOOL_DATA[1]
; --------------------------
PTP {A1 -91.61000,A2 -62.00000,A3 116.14000,A4 -7.59000,A5 -57.42000,A6 5.89000}
; ---- Setting reference (Base) ----
$BASE = {FRAME: X 0.000,Y 0.000,Z 0.000,A 0.000,B 0.000,C 0.000}
; --------------------------
; ---- Setting tool (TCP) ----
; TOOL_DATA[1] = {FRAME: X 0.000,Y 0.000,Z 10.000,A 0.000,B 0.000,C 0.000}
$TOOL = {FRAME: X 0.000,Y 0.000,Z 10.000,A 0.000,B 0.000,C 0.000}
; $TOOL = TOOL_DATA[1]
; --------------------------
PTP {A1 -92.81350,A2 -61.83030,A3 115.90000,A4 -9.01733,A5 -57.45280,A6 6.73043}
; ---- Setting reference (Base) ----
$BASE = {FRAME: X 0.000,Y 0.000,Z 0.000,A 0.000,B 0.000,C 0.000}
; --------------------------
; ---- Setting tool (TCP) ----
; TOOL_DATA[1] = {FRAME: X 0.000,Y 0.000,Z 10.000,A 0.000,B 0.000,C 0.000}
$TOOL = {FRAME: X 0.000,Y 0.000,Z 10.000,A 0.000,B 0.000,C 0.000}
; $TOOL = TOOL_DATA[1]
; --------------------------
PTP {A1 -97.49790,A2 -59.82320,A3 112.25100,A4 -47.29280,A5 -66.19060,A6 26.40350}
; ---- Setting reference (Base) ----
$BASE = {FRAME: X 0.000,Y 0.000,Z 0.000,A 0.000,B 0.000,C 0.000}
; --------------------------
; ---- Setting tool (TCP) ----
; TOOL_DATA[1] = {FRAME: X 0.000,Y 0.000,Z 10.000,A 0.000,B 0.000,C 0.000}
$TOOL = {FRAME: X 0.000,Y 0.000,Z 10.000,A 0.000,B 0.000,C 0.000}
; $TOOL = TOOL_DATA[1]
; --------------------------
PTP {A1 -87.66640,A2 -61.30810,A3 114.40800,A4 32.39760,A5 -59.63670,A6 -16.00830}
; ---- Setting reference (Base) ----
$BASE = {FRAME: X 0.000,Y 0.000,Z 0.000,A 0.000,B 0.000,C 0.000}
; --------------------------
; ---- Setting tool (TCP) ----
; TOOL_DATA[1] = {FRAME: X 0.000,Y 0.000,Z 10.000,A 0.000,B 0.000,C 0.000}
$TOOL = {FRAME: X 0.000,Y 0.000,Z 10.000,A 0.000,B 0.000,C 0.000}
; $TOOL = TOOL_DATA[1]
; --------------------------
PTP {A1 -92.81350,A2 -61.83030,A3 115.90000,A4 -9.01733,A5 -57.45280,A6 6.73043}
; ---- Setting reference (Base) ----
$BASE = {FRAME: X 0.000,Y 0.000,Z 0.000,A 0.000,B 0.000,C 0.000}
; --------------------------
; ---- Setting tool (TCP) ----
; TOOL_DATA[1] = {FRAME: X 0.000,Y 0.000,Z 10.000,A 0.000,B 0.000,C 0.000}
$TOOL = {FRAME: X 0.000,Y 0.000,Z 10.000,A 0.000,B 0.000,C 0.000}
; $TOOL = TOOL_DATA[1]
; --------------------------
PTP {A1 -92.81350,A2 -61.83030,A3 115.90000,A4 -9.01733,A5 -57.45280,A6 -23.26960}
; ---- Setting reference (Base) ----
$BASE = {FRAME: X 0.000,Y 0.000,Z 0.000,A 0.000,B 0.000,C 0.000}
; --------------------------
; ---- Setting tool (TCP) ----
; TOOL_DATA[1] = {FRAME: X 0.000,Y 0.000,Z 10.000,A 0.000,B 0.000,C 0.000}
$TOOL = {FRAME: X 0.000,Y 0.000,Z 10.000,A 0.000,B 0.000,C 0.000}
; $TOOL = TOOL_DATA[1]
; --------------------------
PTP {A1 -92.81350,A2 -61.83030,A3 115.90000,A4 -9.01733,A5 -57.45280,A6 36.73040}
; ---- Setting reference (Base) ----
$BASE = {FRAME: X 0.000,Y 0.000,Z 0.000,A 0.000,B 0.000,C 0.000}
; --------------------------
; ---- Setting tool (TCP) ----
; TOOL_DATA[1] = {FRAME: X 0.000,Y 0.000,Z 10.000,A 0.000,B 0.000,C 0.000}
$TOOL = {FRAME: X 0.000,Y 0.000,Z 10.000,A 0.000,B 0.000,C 0.000}
; $TOOL = TOOL_DATA[1]
; --------------------------
PTP {A1 -92.81350,A2 -61.83030,A3 115.90000,A4 -9.01733,A5 -57.45280,A6 6.73043}
; ---- Setting reference (Base) ----
$BASE = {FRAME: X 0.000,Y 0.000,Z 0.000,A 0.000,B 0.000,C 0.000}
; --------------------------
; ---- Setting tool (TCP) ----
; TOOL_DATA[1] = {FRAME: X 0.000,Y 0.000,Z 10.000,A 0.000,B 0.000,C 0.000}
$TOOL = {FRAME: X 0.000,Y 0.000,Z 10.000,A 0.000,B 0.000,C 0.000}
; $TOOL = TOOL_DATA[1]
; --------------------------
PTP {A1 -94.01030,A2 -61.63900,A3 115.62000,A4 -10.43750,A5 -57.48330,A6 7.57021}
; ---- Setting reference (Base) ----
$BASE = {FRAME: X 0.000,Y 0.000,Z 0.000,A 0.000,B 0.000,C 0.000}
; --------------------------
; ---- Setting tool (TCP) ----
; TOOL_DATA[1] = {FRAME: X 0.000,Y 0.000,Z 10.000,A 0.000,B 0.000,C 0.000}
$TOOL = {FRAME: X 0.000,Y 0.000,Z 10.000,A 0.000,B 0.000,C 0.000}
; $TOOL = TOOL_DATA[1]
; --------------------------
PTP {A1 -98.63160,A2 -59.54800,A3 111.80400,A4 -48.44910,A5 -66.58900,A6 27.04970}
; ---- Setting reference (Base) ----
$BASE = {FRAME: X 0.000,Y 0.000,Z 0.000,A 0.000,B 0.000,C 0.000}
; --------------------------
; ---- Setting tool (TCP) ----
; TOOL_DATA[1] = {FRAME: X 0.000,Y 0.000,Z 10.000,A 0.000,B 0.000,C 0.000}
$TOOL = {FRAME: X 0.000,Y 0.000,Z 10.000,A 0.000,B 0.000,C 0.000}
; $TOOL = TOOL_DATA[1]
; --------------------------
PTP {A1 -88.85630,A2 -61.21070,A3 114.30300,A4 31.08980,A5 -59.25410,A6 -15.30750}
; ---- Setting reference (Base) ----
$BASE = {FRAME: X 0.000,Y 0.000,Z 0.000,A 0.000,B 0.000,C 0.000}
; --------------------------
; ---- Setting tool (TCP) ----
; TOOL_DATA[1] = {FRAME: X 0.000,Y 0.000,Z 10.000,A 0.000,B 0.000,C 0.000}
$TOOL = {FRAME: X 0.000,Y 0.000,Z 10.000,A 0.000,B 0.000,C 0.000}
; $TOOL = TOOL_DATA[1]
; --------------------------
PTP {A1 -94.01030,A2 -61.63900,A3 115.62000,A4 -10.43750,A5 -57.48330,A6 7.57021}
; ---- Setting reference (Base) ----
$BASE = {FRAME: X 0.000,Y 0.000,Z 0.000,A 0.000,B 0.000,C 0.000}
; --------------------------
; ---- Setting tool (TCP) ----
; TOOL_DATA[1] = {FRAME: X 0.000,Y 0.000,Z 10.000,A 0.000,B 0.000,C 0.000}
$TOOL = {FRAME: X 0.000,Y 0.000,Z 10.000,A 0.000,B 0.000,C 0.000}
; $TOOL = TOOL_DATA[1]
; --------------------------
PTP {A1 -94.01030,A2 -61.63900,A3 115.62000,A4 -10.43750,A5 -57.48330,A6 -22.42980}
; ---- Setting reference (Base) ----
$BASE = {FRAME: X 0.000,Y 0.000,Z 0.000,A 0.000,B 0.000,C 0.000}
; --------------------------
; ---- Setting tool (TCP) ----
; TOOL_DATA[1] = {FRAME: X 0.000,Y 0.000,Z 10.000,A 0.000,B 0.000,C 0.000}
$TOOL = {FRAME: X 0.000,Y 0.000,Z 10.000,A 0.000,B 0.000,C 0.000}
; $TOOL = TOOL_DATA[1]
; --------------------------
PTP {A1 -94.01030,A2 -61.63900,A3 115.62000,A4 -10.43750,A5 -57.48330,A6 37.57020}
; ---- Setting reference (Base) ----
$BASE = {FRAME: X 0.000,Y 0.000,Z 0.000,A 0.000,B 0.000,C 0.000}
; --------------------------
; ---- Setting tool (TCP) ----
; TOOL_DATA[1] = {FRAME: X 0.000,Y 0.000,Z 10.000,A 0.000,B 0.000,C 0.000}
$TOOL = {FRAME: X 0.000,Y 0.000,Z 10.000,A 0.000,B 0.000,C 0.000}
; $TOOL = TOOL_DATA[1]
; --------------------------
PTP {A1 -94.01030,A2 -61.63900,A3 115.62000,A4 -10.43750,A5 -57.48330,A6 7.57021}
; ---- Setting reference (Base) ----
$BASE = {FRAME: X 0.000,Y 0.000,Z 0.000,A 0.000,B 0.000,C 0.000}
; --------------------------
; ---- Setting tool (TCP) ----
; TOOL_DATA[1] = {FRAME: X 0.000,Y 0.000,Z 10.000,A 0.000,B 0.000,C 0.000}
$TOOL = {FRAME: X 0.000,Y 0.000,Z 10.000,A 0.000,B 0.000,C 0.000}
; $TOOL = TOOL_DATA[1]
; --------------------------
PTP {A1 -95.19930,A2 -61.42650,A3 115.29800,A4 -11.84960,A5 -57.51140,A6 8.40973}
; ---- Setting reference (Base) ----
$BASE = {FRAME: X 0.000,Y 0.000,Z 0.000,A 0.000,B 0.000,C 0.000}
; --------------------------
; ---- Setting tool (TCP) ----
; TOOL_DATA[1] = {FRAME: X 0.000,Y 0.000,Z 10.000,A 0.000,B 0.000,C 0.000}
$TOOL = {FRAME: X 0.000,Y 0.000,Z 10.000,A 0.000,B 0.000,C 0.000}
; $TOOL = TOOL_DATA[1]
; --------------------------
PTP {A1 -99.75460,A2 -59.25260,A3 111.31800,A4 -49.59170,A5 -66.98360,A6 27.69850}
; ---- Setting reference (Base) ----
$BASE = {FRAME: X 0.000,Y 0.000,Z 0.000,A 0.000,B 0.000,C 0.000}
; --------------------------
; ---- Setting tool (TCP) ----
; TOOL_DATA[1] = {FRAME: X 0.000,Y 0.000,Z 10.000,A 0.000,B 0.000,C 0.000}
$TOOL = {FRAME: X 0.000,Y 0.000,Z 10.000,A 0.000,B 0.000,C 0.000}
; $TOOL = TOOL_DATA[1]
; --------------------------
PTP {A1 -90.04300,A2 -61.09150,A3 114.15600,A4 29.78100,A5 -58.86940,A6 -14.60710}
; ---- Setting reference (Base) ----
$BASE = {FRAME: X 0.000,Y 0.000,Z 0.000,A 0.000,B 0.000,C 0.000}
; --------------------------
; ---- Setting tool (TCP) ----
; TOOL_DATA[1] = {FRAME: X 0.000,Y 0.000,Z 10.000,A 0.000,B 0.000,C 0.000}
$TOOL = {FRAME: X 0.000,Y 0.000,Z 10.000,A 0.000,B 0.000,C 0.000}
; $TOOL = TOOL_DATA[1]
; --------------------------
PTP {A1 -95.19930,A2 -61.42650,A3 115.29800,A4 -11.84960,A5 -57.51140,A6 8.40973}
; ---- Setting reference (Base) ----
$BASE = {FRAME: X 0.000,Y 0.000,Z 0.000,A 0.000,B 0.000,C 0.000}
; --------------------------
; ---- Setting tool (TCP) ----
; TOOL_DATA[1] = {FRAME: X 0.000,Y 0.000,Z 10.000,A 0.000,B 0.000,C 0.000}
$TOOL = {FRAME: X 0.000,Y 0.000,Z 10.000,A 0.000,B 0.000,C 0.000}
; $TOOL = TOOL_DATA[1]
; --------------------------
PTP {A1 -95.19930,A2 -61.42650,A3 115.29800,A4 -11.84960,A5 -57.51140,A6 -21.59030}
; ---- Setting reference (Base) ----
$BASE = {FRAME: X 0.000,Y 0.000,Z 0.000,A 0.000,B 0.000,C 0.000}
; --------------------------
; ---- Setting tool (TCP) ----
; TOOL_DATA[1] = {FRAME: X 0.000,Y 0.000,Z 10.000,A 0.000,B 0.000,C 0.000}
$TOOL = {FRAME: X 0.000,Y 0.000,Z 10.000,A 0.000,B 0.000,C 0.000}
; $TOOL = TOOL_DATA[1]
; --------------------------
PTP {A1 -95.19930,A2 -61.42650,A3 115.29800,A4 -11.84960,A5 -57.51140,A6 38.40970}
; ---- Setting reference (Base) ----
$BASE = {FRAME: X 0.000,Y 0.000,Z 0.000,A 0.000,B 0.000,C 0.000}
; --------------------------
; ---- Setting tool (TCP) ----
; TOOL_DATA[1] = {FRAME: X 0.000,Y 0.000,Z 10.000,A 0.000,B 0.000,C 0.000}
$TOOL = {FRAME: X 0.000,Y 0.000,Z 10.000,A 0.000,B 0.000,C 0.000}
; $TOOL = TOOL_DATA[1]
; --------------------------
PTP {A1 -95.19930,A2 -61.42650,A3 115.29800,A4 -11.84960,A5 -57.51140,A6 8.40973}
; ---- Setting reference (Base) ----
$BASE = {FRAME: X 0.000,Y 0.000,Z 0.000,A 0.000,B 0.000,C 0.000}
; --------------------------
; ---- Setting tool (TCP) ----
; TOOL_DATA[1] = {FRAME: X 0.000,Y 0.000,Z 10.000,A 0.000,B 0.000,C 0.000}
$TOOL = {FRAME: X 0.000,Y 0.000,Z 10.000,A 0.000,B 0.000,C 0.000}
; $TOOL = TOOL_DATA[1]
; --------------------------
PTP {A1 -96.37960,A2 -61.19280,A3 114.93500,A4 -13.25300,A5 -57.53700,A6 9.24939}
; ---- Setting reference (Base) ----
$BASE = {FRAME: X 0.000,Y 0.000,Z 0.000,A 0.000,B 0.000,C 0.000}
; --------------------------
; ---- Setting tool (TCP) ----
; TOOL_DATA[1] = {FRAME: X 0.000,Y 0.000,Z 10.000,A 0.000,B 0.000,C 0.000}
$TOOL = {FRAME: X 0.000,Y 0.000,Z 10.000,A 0.000,B 0.000,C 0.000}
; $TOOL = TOOL_DATA[1]
; --------------------------
PTP {A1 -100.86600,A2 -58.93720,A3 110.79100,A4 -50.72010,A5 -67.37440,A6 28.35040}
; ---- Setting reference (Base) ----
$BASE = {FRAME: X 0.000,Y 0.000,Z 0.000,A 0.000,B 0.000,C 0.000}
; --------------------------
; ---- Setting tool (TCP) ----
; TOOL_DATA[1] = {FRAME: X 0.000,Y 0.000,Z 10.000,A 0.000,B 0.000,C 0.000}
$TOOL = {FRAME: X 0.000,Y 0.000,Z 10.000,A 0.000,B 0.000,C 0.000}
; $TOOL = TOOL_DATA[1]
; --------------------------
PTP {A1 -91.22550,A2 -60.95060,A3 113.96900,A4 28.47190,A5 -58.48250,A6 -13.90670}
; ---- Setting reference (Base) ----
$BASE = {FRAME: X 0.000,Y 0.000,Z 0.000,A 0.000,B 0.000,C 0.000}
; --------------------------
; ---- Setting tool (TCP) ----
; TOOL_DATA[1] = {FRAME: X 0.000,Y 0.000,Z 10.000,A 0.000,B 0.000,C 0.000}
$TOOL = {FRAME: X 0.000,Y 0.000,Z 10.000,A 0.000,B 0.000,C 0.000}
; $TOOL = TOOL_DATA[1]
; --------------------------
PTP {A1 -96.37960,A2 -61.19280,A3 114.93500,A4 -13.25300,A5 -57.53700,A6 9.24939}
; ---- Setting reference (Base) ----
$BASE = {FRAME: X 0.000,Y 0.000,Z 0.000,A 0.000,B 0.000,C 0.000}
; --------------------------
; ---- Setting tool (TCP) ----
; TOOL_DATA[1] = {FRAME: X 0.000,Y 0.000,Z 10.000,A 0.000,B 0.000,C 0.000}
$TOOL = {FRAME: X 0.000,Y 0.000,Z 10.000,A 0.000,B 0.000,C 0.000}
; $TOOL = TOOL_DATA[1]
; --------------------------
PTP {A1 -96.37960,A2 -61.19280,A3 114.93500,A4 -13.25300,A5 -57.53700,A6 -20.75060}
; ---- Setting reference (Base) ----
$BASE = {FRAME: X 0.000,Y 0.000,Z 0.000,A 0.000,B 0.000,C 0.000}
; --------------------------
; ---- Setting tool (TCP) ----
; TOOL_DATA[1] = {FRAME: X 0.000,Y 0.000,Z 10.000,A 0.000,B 0.000,C 0.000}
$TOOL = {FRAME: X 0.000,Y 0.000,Z 10.000,A 0.000,B 0.000,C 0.000}
; $TOOL = TOOL_DATA[1]
; --------------------------
PTP {A1 -96.37960,A2 -61.19280,A3 114.93500,A4 -13.25300,A5 -57.53700,A6 39.24940}
; ---- Setting reference (Base) ----
$BASE = {FRAME: X 0.000,Y 0.000,Z 0.000,A 0.000,B 0.000,C 0.000}
; --------------------------
; ---- Setting tool (TCP) ----
; TOOL_DATA[1] = {FRAME: X 0.000,Y 0.000,Z 10.000,A 0.000,B 0.000,C 0.000}
$TOOL = {FRAME: X 0.000,Y 0.000,Z 10.000,A 0.000,B 0.000,C 0.000}
; $TOOL = TOOL_DATA[1]
; --------------------------
PTP {A1 -96.37960,A2 -61.19280,A3 114.93500,A4 -13.25300,A5 -57.53700,A6 9.24939}
; ---- Setting reference (Base) ----
$BASE = {FRAME: X 0.000,Y 0.000,Z 0.000,A 0.000,B 0.000,C 0.000}
; --------------------------
; ---- Setting tool (TCP) ----
; TOOL_DATA[1] = {FRAME: X 0.000,Y 0.000,Z 10.000,A 0.000,B 0.000,C 0.000}
$TOOL = {FRAME: X 0.000,Y 0.000,Z 10.000,A 0.000,B 0.000,C 0.000}
; $TOOL = TOOL_DATA[1]
; --------------------------
PTP {A1 -85.49590,A2 -60.82240,A3 116.69600,A4 -0.33249,A5 -58.90590,A6 1.63284}
; ---- Setting reference (Base) ----
$BASE = {FRAME: X 0.000,Y 0.000,Z 0.000,A 0.000,B 0.000,C 0.000}
; --------------------------
; ---- Setting tool (TCP) ----
; TOOL_DATA[1] = {FRAME: X 0.000,Y 0.000,Z 10.000,A 0.000,B 0.000,C 0.000}
$TOOL = {FRAME: X 0.000,Y 0.000,Z 10.000,A 0.000,B 0.000,C 0.000}
; $TOOL = TOOL_DATA[1]
; --------------------------
PTP {A1 -90.48090,A2 -59.40400,A3 114.06600,A4 -39.57220,A5 -64.94390,A6 21.39460}
; ---- Setting reference (Base) ----
$BASE = {FRAME: X 0.000,Y 0.000,Z 0.000,A 0.000,B 0.000,C 0.000}
; --------------------------
; ---- Setting tool (TCP) ----
; TOOL_DATA[1] = {FRAME: X 0.000,Y 0.000,Z 10.000,A 0.000,B 0.000,C 0.000}
$TOOL = {FRAME: X 0.000,Y 0.000,Z 10.000,A 0.000,B 0.000,C 0.000}
; $TOOL = TOOL_DATA[1]
; --------------------------
PTP {A1 -80.49230,A2 -59.79470,A3 114.15700,A4 39.65230,A5 -63.15200,A6 -19.07170}
; ---- Setting reference (Base) ----
$BASE = {FRAME: X 0.000,Y 0.000,Z 0.000,A 0.000,B 0.000,C 0.000}
; --------------------------
; ---- Setting tool (TCP) ----
; TOOL_DATA[1] = {FRAME: X 0.000,Y 0.000,Z 10.000,A 0.000,B 0.000,C 0.000}
$TOOL = {FRAME: X 0.000,Y 0.000,Z 10.000,A 0.000,B 0.000,C 0.000}
; $TOOL = TOOL_DATA[1]
; --------------------------
PTP {A1 -85.49590,A2 -60.82240,A3 116.69600,A4 -0.33249,A5 -58.90590,A6 1.63284}
; ---- Setting reference (Base) ----
$BASE = {FRAME: X 0.000,Y 0.000,Z 0.000,A 0.000,B 0.000,C 0.000}
; --------------------------
; ---- Setting tool (TCP) ----
; TOOL_DATA[1] = {FRAME: X 0.000,Y 0.000,Z 10.000,A 0.000,B 0.000,C 0.000}
$TOOL = {FRAME: X 0.000,Y 0.000,Z 10.000,A 0.000,B 0.000,C 0.000}
; $TOOL = TOOL_DATA[1]
; --------------------------
PTP {A1 -85.49590,A2 -60.82240,A3 116.69600,A4 -0.33249,A5 -58.90590,A6 -28.36720}
; ---- Setting reference (Base) ----
$BASE = {FRAME: X 0.000,Y 0.000,Z 0.000,A 0.000,B 0.000,C 0.000}
; --------------------------
; ---- Setting tool (TCP) ----
; TOOL_DATA[1] = {FRAME: X 0.000,Y 0.000,Z 10.000,A 0.000,B 0.000,C 0.000}
$TOOL = {FRAME: X 0.000,Y 0.000,Z 10.000,A 0.000,B 0.000,C 0.000}
; $TOOL = TOOL_DATA[1]
; --------------------------
PTP {A1 -85.49590,A2 -60.82240,A3 116.69600,A4 -0.33249,A5 -58.90590,A6 31.63280}
; ---- Setting reference (Base) ----
$BASE = {FRAME: X 0.000,Y 0.000,Z 0.000,A 0.000,B 0.000,C 0.000}
; --------------------------
; ---- Setting tool (TCP) ----
; TOOL_DATA[1] = {FRAME: X 0.000,Y 0.000,Z 10.000,A 0.000,B 0.000,C 0.000}
$TOOL = {FRAME: X 0.000,Y 0.000,Z 10.000,A 0.000,B 0.000,C 0.000}
; $TOOL = TOOL_DATA[1]
; --------------------------
PTP {A1 -85.49590,A2 -60.82240,A3 116.69600,A4 -0.33249,A5 -58.90590,A6 1.63284}
; ---- Setting reference (Base) ----
$BASE = {FRAME: X 0.000,Y 0.000,Z 0.000,A 0.000,B 0.000,C 0.000}
; --------------------------
; ---- Setting tool (TCP) ----
; TOOL_DATA[1] = {FRAME: X 0.000,Y 0.000,Z 10.000,A 0.000,B 0.000,C 0.000}
$TOOL = {FRAME: X 0.000,Y 0.000,Z 10.000,A 0.000,B 0.000,C 0.000}
; $TOOL = TOOL_DATA[1]
; --------------------------
PTP {A1 -86.71630,A2 -60.76350,A3 116.66400,A4 -1.75494,A5 -58.94530,A6 2.43120}
; ---- Setting reference (Base) ----
$BASE = {FRAME: X 0.000,Y 0.000,Z 0.000,A 0.000,B 0.000,C 0.000}
; --------------------------
; ---- Setting tool (TCP) ----
; TOOL_DATA[1] = {FRAME: X 0.000,Y 0.000,Z 10.000,A 0.000,B 0.000,C 0.000}
$TOOL = {FRAME: X 0.000,Y 0.000,Z 10.000,A 0.000,B 0.000,C 0.000}
; $TOOL = TOOL_DATA[1]
; --------------------------
PTP {A1 -91.66030,A2 -59.25910,A3 113.86200,A4 -40.79340,A5 -65.33890,A6 22.01180}
; ---- Setting reference (Base) ----
$BASE = {FRAME: X 0.000,Y 0.000,Z 0.000,A 0.000,B 0.000,C 0.000}
; --------------------------
; ---- Setting tool (TCP) ----
; TOOL_DATA[1] = {FRAME: X 0.000,Y 0.000,Z 10.000,A 0.000,B 0.000,C 0.000}
$TOOL = {FRAME: X 0.000,Y 0.000,Z 10.000,A 0.000,B 0.000,C 0.000}
; $TOOL = TOOL_DATA[1]
; --------------------------
PTP {A1 -81.67850,A2 -59.82650,A3 114.29900,A4 38.37880,A5 -62.80290,A6 -18.39190}
; ---- Setting reference (Base) ----
$BASE = {FRAME: X 0.000,Y 0.000,Z 0.000,A 0.000,B 0.000,C 0.000}
; --------------------------
; ---- Setting tool (TCP) ----
; TOOL_DATA[1] = {FRAME: X 0.000,Y 0.000,Z 10.000,A 0.000,B 0.000,C 0.000}
$TOOL = {FRAME: X 0.000,Y 0.000,Z 10.000,A 0.000,B 0.000,C 0.000}
; $TOOL = TOOL_DATA[1]
; --------------------------
PTP {A1 -86.71630,A2 -60.76350,A3 116.66400,A4 -1.75494,A5 -58.94530,A6 2.43120}
; ---- Setting reference (Base) ----
$BASE = {FRAME: X 0.000,Y 0.000,Z 0.000,A 0.000,B 0.000,C 0.000}
; --------------------------
; ---- Setting tool (TCP) ----
; TOOL_DATA[1] = {FRAME: X 0.000,Y 0.000,Z 10.000,A 0.000,B 0.000,C 0.000}
$TOOL = {FRAME: X 0.000,Y 0.000,Z 10.000,A 0.000,B 0.000,C 0.000}
; $TOOL = TOOL_DATA[1]
; --------------------------
PTP {A1 -86.71630,A2 -60.76350,A3 116.66400,A4 -1.75494,A5 -58.94530,A6 -27.56880}
; ---- Setting reference (Base) ----
$BASE = {FRAME: X 0.000,Y 0.000,Z 0.000,A 0.000,B 0.000,C 0.000}
; --------------------------
; ---- Setting tool (TCP) ----
; TOOL_DATA[1] = {FRAME: X 0.000,Y 0.000,Z 10.000,A 0.000,B 0.000,C 0.000}
$TOOL = {FRAME: X 0.000,Y 0.000,Z 10.000,A 0.000,B 0.000,C 0.000}
; $TOOL = TOOL_DATA[1]
; --------------------------
PTP {A1 -86.71630,A2 -60.76350,A3 116.66400,A4 -1.75494,A5 -58.94530,A6 32.43120}
; ---- Setting reference (Base) ----
$BASE = {FRAME: X 0.000,Y 0.000,Z 0.000,A 0.000,B 0.000,C 0.000}
; --------------------------
; ---- Setting tool (TCP) ----
; TOOL_DATA[1] = {FRAME: X 0.000,Y 0.000,Z 10.000,A 0.000,B 0.000,C 0.000}
$TOOL = {FRAME: X 0.000,Y 0.000,Z 10.000,A 0.000,B 0.000,C 0.000}
; $TOOL = TOOL_DATA[1]
; --------------------------
PTP {A1 -86.71630,A2 -60.76350,A3 116.66400,A4 -1.75494,A5 -58.94530,A6 2.43120}
; ---- Setting reference (Base) ----
$BASE = {FRAME: X 0.000,Y 0.000,Z 0.000,A 0.000,B 0.000,C 0.000}
; --------------------------
; ---- Setting tool (TCP) ----
; TOOL_DATA[1] = {FRAME: X 0.000,Y 0.000,Z 10.000,A 0.000,B 0.000,C 0.000}
$TOOL = {FRAME: X 0.000,Y 0.000,Z 10.000,A 0.000,B 0.000,C 0.000}
; $TOOL = TOOL_DATA[1]
; --------------------------
PTP {A1 -87.93520,A2 -60.68340,A3 116.59000,A4 -3.17495,A5 -58.98120,A6 3.22760}
; ---- Setting reference (Base) ----
$BASE = {FRAME: X 0.000,Y 0.000,Z 0.000,A 0.000,B 0.000,C 0.000}
; --------------------------
; ---- Setting tool (TCP) ----
; TOOL_DATA[1] = {FRAME: X 0.000,Y 0.000,Z 10.000,A 0.000,B 0.000,C 0.000}
$TOOL = {FRAME: X 0.000,Y 0.000,Z 10.000,A 0.000,B 0.000,C 0.000}
; $TOOL = TOOL_DATA[1]
; --------------------------
PTP {A1 -92.83410,A2 -59.09360,A3 113.61700,A4 -42.00620,A5 -65.72910,A6 22.63070}
; ---- Setting reference (Base) ----
$BASE = {FRAME: X 0.000,Y 0.000,Z 0.000,A 0.000,B 0.000,C 0.000}
; --------------------------
; ---- Setting tool (TCP) ----
; TOOL_DATA[1] = {FRAME: X 0.000,Y 0.000,Z 10.000,A 0.000,B 0.000,C 0.000}
$TOOL = {FRAME: X 0.000,Y 0.000,Z 10.000,A 0.000,B 0.000,C 0.000}
; $TOOL = TOOL_DATA[1]
; --------------------------
PTP {A1 -82.86760,A2 -59.83700,A3 114.40000,A4 37.09930,A5 -62.45170,A6 -17.71510}
; ---- Setting reference (Base) ----
$BASE = {FRAME: X 0.000,Y 0.000,Z 0.000,A 0.000,B 0.000,C 0.000}
; --------------------------
; ---- Setting tool (TCP) ----
; TOOL_DATA[1] = {FRAME: X 0.000,Y 0.000,Z 10.000,A 0.000,B 0.000,C 0.000}
$TOOL = {FRAME: X 0.000,Y 0.000,Z 10.000,A 0.000,B 0.000,C 0.000}
; $TOOL = TOOL_DATA[1]
; --------------------------
PTP {A1 -87.93520,A2 -60.68340,A3 116.59000,A4 -3.17495,A5 -58.98120,A6 3.22760}
; ---- Setting reference (Base) ----
$BASE = {FRAME: X 0.000,Y 0.000,Z 0.000,A 0.000,B 0.000,C 0.000}
; --------------------------
; ---- Setting tool (TCP) ----
; TOOL_DATA[1] = {FRAME: X 0.000,Y 0.000,Z 10.000,A 0.000,B 0.000,C 0.000}
$TOOL = {FRAME: X 0.000,Y 0.000,Z 10.000,A 0.000,B 0.000,C 0.000}
; $TOOL = TOOL_DATA[1]
; --------------------------
PTP {A1 -87.93520,A2 -60.68340,A3 116.59000,A4 -3.17495,A5 -58.98120,A6 -26.77240}
; ---- Setting reference (Base) ----
$BASE = {FRAME: X 0.000,Y 0.000,Z 0.000,A 0.000,B 0.000,C 0.000}
; --------------------------
; ---- Setting tool (TCP) ----
; TOOL_DATA[1] = {FRAME: X 0.000,Y 0.000,Z 10.000,A 0.000,B 0.000,C 0.000}
$TOOL = {FRAME: X 0.000,Y 0.000,Z 10.000,A 0.000,B 0.000,C 0.000}
; $TOOL = TOOL_DATA[1]
; --------------------------
PTP {A1 -87.93520,A2 -60.68340,A3 116.59000,A4 -3.17495,A5 -58.98120,A6 33.22760}
; ---- Setting reference (Base) ----
$BASE = {FRAME: X 0.000,Y 0.000,Z 0.000,A 0.000,B 0.000,C 0.000}
; --------------------------
; ---- Setting tool (TCP) ----
; TOOL_DATA[1] = {FRAME: X 0.000,Y 0.000,Z 10.000,A 0.000,B 0.000,C 0.000}
$TOOL = {FRAME: X 0.000,Y 0.000,Z 10.000,A 0.000,B 0.000,C 0.000}
; $TOOL = TOOL_DATA[1]
; --------------------------
PTP {A1 -87.93520,A2 -60.68340,A3 116.59000,A4 -3.17495,A5 -58.98120,A6 3.22760}
; ---- Setting reference (Base) ----
$BASE = {FRAME: X 0.000,Y 0.000,Z 0.000,A 0.000,B 0.000,C 0.000}
; --------------------------
; ---- Setting tool (TCP) ----
; TOOL_DATA[1] = {FRAME: X 0.000,Y 0.000,Z 10.000,A 0.000,B 0.000,C 0.000}
$TOOL = {FRAME: X 0.000,Y 0.000,Z 10.000,A 0.000,B 0.000,C 0.000}
; $TOOL = TOOL_DATA[1]
; --------------------------
PTP {A1 -89.15160,A2 -60.58220,A3 116.47500,A4 -4.59164,A5 -59.01330,A6 4.02249}
; ---- Setting reference (Base) ----
$BASE = {FRAME: X 0.000,Y 0.000,Z 0.000,A 0.000,B 0.000,C 0.000}
; --------------------------
; ---- Setting tool (TCP) ----
; TOOL_DATA[1] = {FRAME: X 0.000,Y 0.000,Z 10.000,A 0.000,B 0.000,C 0.000}
$TOOL = {FRAME: X 0.000,Y 0.000,Z 10.000,A 0.000,B 0.000,C 0.000}
; $TOOL = TOOL_DATA[1]
; --------------------------
PTP {A1 -94.00150,A2 -58.90780,A3 113.33000,A4 -43.20970,A5 -66.11450,A6 23.25200}
; ---- Setting reference (Base) ----
$BASE = {FRAME: X 0.000,Y 0.000,Z 0.000,A 0.000,B 0.000,C 0.000}
; --------------------------
; ---- Setting tool (TCP) ----
; TOOL_DATA[1] = {FRAME: X 0.000,Y 0.000,Z 10.000,A 0.000,B 0.000,C 0.000}
$TOOL = {FRAME: X 0.000,Y 0.000,Z 10.000,A 0.000,B 0.000,C 0.000}
; $TOOL = TOOL_DATA[1]
; --------------------------
PTP {A1 -84.05880,A2 -59.82630,A3 114.45900,A4 35.81480,A5 -62.09800,A6 -17.04110}
; ---- Setting reference (Base) ----
$BASE = {FRAME: X 0.000,Y 0.000,Z 0.000,A 0.000,B 0.000,C 0.000}
; --------------------------
; ---- Setting tool (TCP) ----
; TOOL_DATA[1] = {FRAME: X 0.000,Y 0.000,Z 10.000,A 0.000,B 0.000,C 0.000}
$TOOL = {FRAME: X 0.000,Y 0.000,Z 10.000,A 0.000,B 0.000,C 0.000}
; $TOOL = TOOL_DATA[1]
; --------------------------
PTP {A1 -89.15160,A2 -60.58220,A3 116.47500,A4 -4.59164,A5 -59.01330,A6 4.02249}
; ---- Setting reference (Base) ----
$BASE = {FRAME: X 0.000,Y 0.000,Z 0.000,A 0.000,B 0.000,C 0.000}
; --------------------------
; ---- Setting tool (TCP) ----
; TOOL_DATA[1] = {FRAME: X 0.000,Y 0.000,Z 10.000,A 0.000,B 0.000,C 0.000}
$TOOL = {FRAME: X 0.000,Y 0.000,Z 10.000,A 0.000,B 0.000,C 0.000}
; $TOOL = TOOL_DATA[1]
; --------------------------
PTP {A1 -89.15160,A2 -60.58220,A3 116.47500,A4 -4.59164,A5 -59.01330,A6 -25.97750}
; ---- Setting reference (Base) ----
$BASE = {FRAME: X 0.000,Y 0.000,Z 0.000,A 0.000,B 0.000,C 0.000}
; --------------------------
; ---- Setting tool (TCP) ----
; TOOL_DATA[1] = {FRAME: X 0.000,Y 0.000,Z 10.000,A 0.000,B 0.000,C 0.000}
$TOOL = {FRAME: X 0.000,Y 0.000,Z 10.000,A 0.000,B 0.000,C 0.000}
; $TOOL = TOOL_DATA[1]
; --------------------------
PTP {A1 -89.15160,A2 -60.58220,A3 116.47500,A4 -4.59164,A5 -59.01330,A6 34.02250}
; ---- Setting reference (Base) ----
$BASE = {FRAME: X 0.000,Y 0.000,Z 0.000,A 0.000,B 0.000,C 0.000}
; --------------------------
; ---- Setting tool (TCP) ----
; TOOL_DATA[1] = {FRAME: X 0.000,Y 0.000,Z 10.000,A 0.000,B 0.000,C 0.000}
$TOOL = {FRAME: X 0.000,Y 0.000,Z 10.000,A 0.000,B 0.000,C 0.000}
; $TOOL = TOOL_DATA[1]
; --------------------------
PTP {A1 -89.15160,A2 -60.58220,A3 116.47500,A4 -4.59164,A5 -59.01330,A6 4.02249}
; ---- Setting reference (Base) ----
$BASE = {FRAME: X 0.000,Y 0.000,Z 0.000,A 0.000,B 0.000,C 0.000}
; --------------------------
; ---- Setting tool (TCP) ----
; TOOL_DATA[1] = {FRAME: X 0.000,Y 0.000,Z 10.000,A 0.000,B 0.000,C 0.000}
$TOOL = {FRAME: X 0.000,Y 0.000,Z 10.000,A 0.000,B 0.000,C 0.000}
; $TOOL = TOOL_DATA[1]
; --------------------------
PTP {A1 -90.36430,A2 -60.45990,A3 116.31800,A4 -6.00414,A5 -59.04150,A6 4.81633}
; ---- Setting reference (Base) ----
$BASE = {FRAME: X 0.000,Y 0.000,Z 0.000,A 0.000,B 0.000,C 0.000}
; --------------------------
; ---- Setting tool (TCP) ----
; TOOL_DATA[1] = {FRAME: X 0.000,Y 0.000,Z 10.000,A 0.000,B 0.000,C 0.000}
$TOOL = {FRAME: X 0.000,Y 0.000,Z 10.000,A 0.000,B 0.000,C 0.000}
; $TOOL = TOOL_DATA[1]
; --------------------------
PTP {A1 -95.16160,A2 -58.70180,A3 113.00400,A4 -44.40330,A5 -66.49520,A6 23.87590}
; ---- Setting reference (Base) ----
$BASE = {FRAME: X 0.000,Y 0.000,Z 0.000,A 0.000,B 0.000,C 0.000}
; --------------------------
; ---- Setting tool (TCP) ----
; TOOL_DATA[1] = {FRAME: X 0.000,Y 0.000,Z 10.000,A 0.000,B 0.000,C 0.000}
$TOOL = {FRAME: X 0.000,Y 0.000,Z 10.000,A 0.000,B 0.000,C 0.000}
; $TOOL = TOOL_DATA[1]
; --------------------------
PTP {A1 -85.25080,A2 -59.79440,A3 114.47700,A4 34.52630,A5 -61.74170,A6 -16.36960}
; ---- Setting reference (Base) ----
$BASE = {FRAME: X 0.000,Y 0.000,Z 0.000,A 0.000,B 0.000,C 0.000}
; --------------------------
; ---- Setting tool (TCP) ----
; TOOL_DATA[1] = {FRAME: X 0.000,Y 0.000,Z 10.000,A 0.000,B 0.000,C 0.000}
$TOOL = {FRAME: X 0.000,Y 0.000,Z 10.000,A 0.000,B 0.000,C 0.000}
; $TOOL = TOOL_DATA[1]
; --------------------------
PTP {A1 -90.36430,A2 -60.45990,A3 116.31800,A4 -6.00414,A5 -59.04150,A6 4.81633}
; ---- Setting reference (Base) ----
$BASE = {FRAME: X 0.000,Y 0.000,Z 0.000,A 0.000,B 0.000,C 0.000}
; --------------------------
; ---- Setting tool (TCP) ----
; TOOL_DATA[1] = {FRAME: X 0.000,Y 0.000,Z 10.000,A 0.000,B 0.000,C 0.000}
$TOOL = {FRAME: X 0.000,Y 0.000,Z 10.000,A 0.000,B 0.000,C 0.000}
; $TOOL = TOOL_DATA[1]
; --------------------------
PTP {A1 -90.36430,A2 -60.45990,A3 116.31800,A4 -6.00414,A5 -59.04150,A6 -25.18370}
; ---- Setting reference (Base) ----
$BASE = {FRAME: X 0.000,Y 0.000,Z 0.000,A 0.000,B 0.000,C 0.000}
; --------------------------
; ---- Setting tool (TCP) ----
; TOOL_DATA[1] = {FRAME: X 0.000,Y 0.000,Z 10.000,A 0.000,B 0.000,C 0.000}
$TOOL = {FRAME: X 0.000,Y 0.000,Z 10.000,A 0.000,B 0.000,C 0.000}
; $TOOL = TOOL_DATA[1]
; --------------------------
PTP {A1 -90.36430,A2 -60.45990,A3 116.31800,A4 -6.00414,A5 -59.04150,A6 34.81630}
; ---- Setting reference (Base) ----
$BASE = {FRAME: X 0.000,Y 0.000,Z 0.000,A 0.000,B 0.000,C 0.000}
; --------------------------
; ---- Setting tool (TCP) ----
; TOOL_DATA[1] = {FRAME: X 0.000,Y 0.000,Z 10.000,A 0.000,B 0.000,C 0.000}
$TOOL = {FRAME: X 0.000,Y 0.000,Z 10.000,A 0.000,B 0.000,C 0.000}
; $TOOL = TOOL_DATA[1]
; --------------------------
PTP {A1 -90.36430,A2 -60.45990,A3 116.31800,A4 -6.00414,A5 -59.04150,A6 4.81633}
; ---- Setting reference (Base) ----
$BASE = {FRAME: X 0.000,Y 0.000,Z 0.000,A 0.000,B 0.000,C 0.000}
; --------------------------
; ---- Setting tool (TCP) ----
; TOOL_DATA[1] = {FRAME: X 0.000,Y 0.000,Z 10.000,A 0.000,B 0.000,C 0.000}
$TOOL = {FRAME: X 0.000,Y 0.000,Z 10.000,A 0.000,B 0.000,C 0.000}
; $TOOL = TOOL_DATA[1]
; --------------------------
PTP {A1 -91.57240,A2 -60.31670,A3 116.11900,A4 -7.41161,A5 -59.06580,A6 5.60958}
; ---- Setting reference (Base) ----
$BASE = {FRAME: X 0.000,Y 0.000,Z 0.000,A 0.000,B 0.000,C 0.000}
; --------------------------
; ---- Setting tool (TCP) ----
; TOOL_DATA[1] = {FRAME: X 0.000,Y 0.000,Z 10.000,A 0.000,B 0.000,C 0.000}
$TOOL = {FRAME: X 0.000,Y 0.000,Z 10.000,A 0.000,B 0.000,C 0.000}
; $TOOL = TOOL_DATA[1]
; --------------------------
PTP {A1 -96.31340,A2 -58.47570,A3 112.63600,A4 -45.58600,A5 -66.87150,A6 24.50290}
; ---- Setting reference (Base) ----
$BASE = {FRAME: X 0.000,Y 0.000,Z 0.000,A 0.000,B 0.000,C 0.000}
; --------------------------
; ---- Setting tool (TCP) ----
; TOOL_DATA[1] = {FRAME: X 0.000,Y 0.000,Z 10.000,A 0.000,B 0.000,C 0.000}
$TOOL = {FRAME: X 0.000,Y 0.000,Z 10.000,A 0.000,B 0.000,C 0.000}
; $TOOL = TOOL_DATA[1]
; --------------------------
PTP {A1 -86.44280,A2 -59.74130,A3 114.45400,A4 33.23480,A5 -61.38250,A6 -15.70030}
; ---- Setting reference (Base) ----
$BASE = {FRAME: X 0.000,Y 0.000,Z 0.000,A 0.000,B 0.000,C 0.000}
; --------------------------
; ---- Setting tool (TCP) ----
; TOOL_DATA[1] = {FRAME: X 0.000,Y 0.000,Z 10.000,A 0.000,B 0.000,C 0.000}
$TOOL = {FRAME: X 0.000,Y 0.000,Z 10.000,A 0.000,B 0.000,C 0.000}
; $TOOL = TOOL_DATA[1]
; --------------------------
PTP {A1 -91.57240,A2 -60.31670,A3 116.11900,A4 -7.41161,A5 -59.06580,A6 5.60958}
; ---- Setting reference (Base) ----
$BASE = {FRAME: X 0.000,Y 0.000,Z 0.000,A 0.000,B 0.000,C 0.000}
; --------------------------
; ---- Setting tool (TCP) ----
; TOOL_DATA[1] = {FRAME: X 0.000,Y 0.000,Z 10.000,A 0.000,B 0.000,C 0.000}
$TOOL = {FRAME: X 0.000,Y 0.000,Z 10.000,A 0.000,B 0.000,C 0.000}
; $TOOL = TOOL_DATA[1]
; --------------------------
PTP {A1 -91.57240,A2 -60.31670,A3 116.11900,A4 -7.41161,A5 -59.06580,A6 -24.39040}
; ---- Setting reference (Base) ----
$BASE = {FRAME: X 0.000,Y 0.000,Z 0.000,A 0.000,B 0.000,C 0.000}
; --------------------------
; ---- Setting tool (TCP) ----
; TOOL_DATA[1] = {FRAME: X 0.000,Y 0.000,Z 10.000,A 0.000,B 0.000,C 0.000}
$TOOL = {FRAME: X 0.000,Y 0.000,Z 10.000,A 0.000,B 0.000,C 0.000}
; $TOOL = TOOL_DATA[1]
; --------------------------
PTP {A1 -91.57240,A2 -60.31670,A3 116.11900,A4 -7.41161,A5 -59.06580,A6 35.60960}
; ---- Setting reference (Base) ----
$BASE = {FRAME: X 0.000,Y 0.000,Z 0.000,A 0.000,B 0.000,C 0.000}
; --------------------------
; ---- Setting tool (TCP) ----
; TOOL_DATA[1] = {FRAME: X 0.000,Y 0.000,Z 10.000,A 0.000,B 0.000,C 0.000}
$TOOL = {FRAME: X 0.000,Y 0.000,Z 10.000,A 0.000,B 0.000,C 0.000}
; $TOOL = TOOL_DATA[1]
; --------------------------
PTP {A1 -91.57240,A2 -60.31670,A3 116.11900,A4 -7.41161,A5 -59.06580,A6 5.60958}
; ---- Setting reference (Base) ----
$BASE = {FRAME: X 0.000,Y 0.000,Z 0.000,A 0.000,B 0.000,C 0.000}
; --------------------------
; ---- Setting tool (TCP) ----
; TOOL_DATA[1] = {FRAME: X 0.000,Y 0.000,Z 10.000,A 0.000,B 0.000,C 0.000}
$TOOL = {FRAME: X 0.000,Y 0.000,Z 10.000,A 0.000,B 0.000,C 0.000}
; $TOOL = TOOL_DATA[1]
; --------------------------
PTP {A1 -92.77480,A2 -60.15270,A3 115.87900,A4 -8.81326,A5 -59.08590,A6 6.40272}
; ---- Setting reference (Base) ----
$BASE = {FRAME: X 0.000,Y 0.000,Z 0.000,A 0.000,B 0.000,C 0.000}
; --------------------------
; ---- Setting tool (TCP) ----
; TOOL_DATA[1] = {FRAME: X 0.000,Y 0.000,Z 10.000,A 0.000,B 0.000,C 0.000}
$TOOL = {FRAME: X 0.000,Y 0.000,Z 10.000,A 0.000,B 0.000,C 0.000}
; $TOOL = TOOL_DATA[1]
; --------------------------
PTP {A1 -97.45610,A2 -58.22970,A3 112.22900,A4 -46.75720,A5 -67.24330,A6 25.13350}
; ---- Setting reference (Base) ----
$BASE = {FRAME: X 0.000,Y 0.000,Z 0.000,A 0.000,B 0.000,C 0.000}
; --------------------------
; ---- Setting tool (TCP) ----
; TOOL_DATA[1] = {FRAME: X 0.000,Y 0.000,Z 10.000,A 0.000,B 0.000,C 0.000}
$TOOL = {FRAME: X 0.000,Y 0.000,Z 10.000,A 0.000,B 0.000,C 0.000}
; $TOOL = TOOL_DATA[1]
; --------------------------
PTP {A1 -87.63360,A2 -59.66720,A3 114.38900,A4 31.94120,A5 -61.02020,A6 -15.03310}
; ---- Setting reference (Base) ----
$BASE = {FRAME: X 0.000,Y 0.000,Z 0.000,A 0.000,B 0.000,C 0.000}
; --------------------------
; ---- Setting tool (TCP) ----
; TOOL_DATA[1] = {FRAME: X 0.000,Y 0.000,Z 10.000,A 0.000,B 0.000,C 0.000}
$TOOL = {FRAME: X 0.000,Y 0.000,Z 10.000,A 0.000,B 0.000,C 0.000}
; $TOOL = TOOL_DATA[1]
; --------------------------
PTP {A1 -92.77480,A2 -60.15270,A3 115.87900,A4 -8.81326,A5 -59.08590,A6 6.40272}
; ---- Setting reference (Base) ----
$BASE = {FRAME: X 0.000,Y 0.000,Z 0.000,A 0.000,B 0.000,C 0.000}
; --------------------------
; ---- Setting tool (TCP) ----
; TOOL_DATA[1] = {FRAME: X 0.000,Y 0.000,Z 10.000,A 0.000,B 0.000,C 0.000}
$TOOL = {FRAME: X 0.000,Y 0.000,Z 10.000,A 0.000,B 0.000,C 0.000}
; $TOOL = TOOL_DATA[1]
; --------------------------
PTP {A1 -92.77480,A2 -60.15270,A3 115.87900,A4 -8.81326,A5 -59.08590,A6 -23.59730}
; ---- Setting reference (Base) ----
$BASE = {FRAME: X 0.000,Y 0.000,Z 0.000,A 0.000,B 0.000,C 0.000}
; --------------------------
; ---- Setting tool (TCP) ----
; TOOL_DATA[1] = {FRAME: X 0.000,Y 0.000,Z 10.000,A 0.000,B 0.000,C 0.000}
$TOOL = {FRAME: X 0.000,Y 0.000,Z 10.000,A 0.000,B 0.000,C 0.000}
; $TOOL = TOOL_DATA[1]
; --------------------------
PTP {A1 -92.77480,A2 -60.15270,A3 115.87900,A4 -8.81326,A5 -59.08590,A6 36.40270}
; ---- Setting reference (Base) ----
$BASE = {FRAME: X 0.000,Y 0.000,Z 0.000,A 0.000,B 0.000,C 0.000}
; --------------------------
; ---- Setting tool (TCP) ----
; TOOL_DATA[1] = {FRAME: X 0.000,Y 0.000,Z 10.000,A 0.000,B 0.000,C 0.000}
$TOOL = {FRAME: X 0.000,Y 0.000,Z 10.000,A 0.000,B 0.000,C 0.000}
; $TOOL = TOOL_DATA[1]
; --------------------------
PTP {A1 -92.77480,A2 -60.15270,A3 115.87900,A4 -8.81326,A5 -59.08590,A6 6.40272}
; ---- Setting reference (Base) ----
$BASE = {FRAME: X 0.000,Y 0.000,Z 0.000,A 0.000,B 0.000,C 0.000}
; --------------------------
; ---- Setting tool (TCP) ----
; TOOL_DATA[1] = {FRAME: X 0.000,Y 0.000,Z 10.000,A 0.000,B 0.000,C 0.000}
$TOOL = {FRAME: X 0.000,Y 0.000,Z 10.000,A 0.000,B 0.000,C 0.000}
; $TOOL = TOOL_DATA[1]
; --------------------------
PTP {A1 -93.97040,A2 -59.96820,A3 115.59800,A4 -10.20830,A5 -59.10190,A6 7.19624}
; ---- Setting reference (Base) ----
$BASE = {FRAME: X 0.000,Y 0.000,Z 0.000,A 0.000,B 0.000,C 0.000}
; --------------------------
; ---- Setting tool (TCP) ----
; TOOL_DATA[1] = {FRAME: X 0.000,Y 0.000,Z 10.000,A 0.000,B 0.000,C 0.000}
$TOOL = {FRAME: X 0.000,Y 0.000,Z 10.000,A 0.000,B 0.000,C 0.000}
; $TOOL = TOOL_DATA[1]
; --------------------------
PTP {A1 -98.58890,A2 -57.96400,A3 111.78200,A4 -47.91620,A5 -67.61080,A6 25.76800}
; ---- Setting reference (Base) ----
$BASE = {FRAME: X 0.000,Y 0.000,Z 0.000,A 0.000,B 0.000,C 0.000}
; --------------------------
; ---- Setting tool (TCP) ----
; TOOL_DATA[1] = {FRAME: X 0.000,Y 0.000,Z 10.000,A 0.000,B 0.000,C 0.000}
$TOOL = {FRAME: X 0.000,Y 0.000,Z 10.000,A 0.000,B 0.000,C 0.000}
; $TOOL = TOOL_DATA[1]
; --------------------------
PTP {A1 -88.82230,A2 -59.57210,A3 114.28400,A4 30.64660,A5 -60.65440,A6 -14.36750}
; ---- Setting reference (Base) ----
$BASE = {FRAME: X 0.000,Y 0.000,Z 0.000,A 0.000,B 0.000,C 0.000}
; --------------------------
; ---- Setting tool (TCP) ----
; TOOL_DATA[1] = {FRAME: X 0.000,Y 0.000,Z 10.000,A 0.000,B 0.000,C 0.000}
$TOOL = {FRAME: X 0.000,Y 0.000,Z 10.000,A 0.000,B 0.000,C 0.000}
; $TOOL = TOOL_DATA[1]
; --------------------------
PTP {A1 -93.97040,A2 -59.96820,A3 115.59800,A4 -10.20830,A5 -59.10190,A6 7.19624}
; ---- Setting reference (Base) ----
$BASE = {FRAME: X 0.000,Y 0.000,Z 0.000,A 0.000,B 0.000,C 0.000}
; --------------------------
; ---- Setting tool (TCP) ----
; TOOL_DATA[1] = {FRAME: X 0.000,Y 0.000,Z 10.000,A 0.000,B 0.000,C 0.000}
$TOOL = {FRAME: X 0.000,Y 0.000,Z 10.000,A 0.000,B 0.000,C 0.000}
; $TOOL = TOOL_DATA[1]
; --------------------------
PTP {A1 -93.97040,A2 -59.96820,A3 115.59800,A4 -10.20830,A5 -59.10190,A6 -22.80380}
; ---- Setting reference (Base) ----
$BASE = {FRAME: X 0.000,Y 0.000,Z 0.000,A 0.000,B 0.000,C 0.000}
; --------------------------
; ---- Setting tool (TCP) ----
; TOOL_DATA[1] = {FRAME: X 0.000,Y 0.000,Z 10.000,A 0.000,B 0.000,C 0.000}
$TOOL = {FRAME: X 0.000,Y 0.000,Z 10.000,A 0.000,B 0.000,C 0.000}
; $TOOL = TOOL_DATA[1]
; --------------------------
PTP {A1 -93.97040,A2 -59.96820,A3 115.59800,A4 -10.20830,A5 -59.10190,A6 37.19620}
; ---- Setting reference (Base) ----
$BASE = {FRAME: X 0.000,Y 0.000,Z 0.000,A 0.000,B 0.000,C 0.000}
; --------------------------
; ---- Setting tool (TCP) ----
; TOOL_DATA[1] = {FRAME: X 0.000,Y 0.000,Z 10.000,A 0.000,B 0.000,C 0.000}
$TOOL = {FRAME: X 0.000,Y 0.000,Z 10.000,A 0.000,B 0.000,C 0.000}
; $TOOL = TOOL_DATA[1]
; --------------------------
PTP {A1 -93.97040,A2 -59.96820,A3 115.59800,A4 -10.20830,A5 -59.10190,A6 7.19624}
; ---- Setting reference (Base) ----
$BASE = {FRAME: X 0.000,Y 0.000,Z 0.000,A 0.000,B 0.000,C 0.000}
; --------------------------
; ---- Setting tool (TCP) ----
; TOOL_DATA[1] = {FRAME: X 0.000,Y 0.000,Z 10.000,A 0.000,B 0.000,C 0.000}
$TOOL = {FRAME: X 0.000,Y 0.000,Z 10.000,A 0.000,B 0.000,C 0.000}
; $TOOL = TOOL_DATA[1]
; --------------------------
PTP {A1 -95.15830,A2 -59.76330,A3 115.27600,A4 -11.59600,A5 -59.11370,A6 7.99064}
; ---- Setting reference (Base) ----
$BASE = {FRAME: X 0.000,Y 0.000,Z 0.000,A 0.000,B 0.000,C 0.000}
; --------------------------
; ---- Setting tool (TCP) ----
; TOOL_DATA[1] = {FRAME: X 0.000,Y 0.000,Z 10.000,A 0.000,B 0.000,C 0.000}
$TOOL = {FRAME: X 0.000,Y 0.000,Z 10.000,A 0.000,B 0.000,C 0.000}
; $TOOL = TOOL_DATA[1]
; --------------------------
PTP {A1 -99.71110,A2 -57.67880,A3 111.29400,A4 -49.06230,A5 -67.97420,A6 26.40680}
; ---- Setting reference (Base) ----
$BASE = {FRAME: X 0.000,Y 0.000,Z 0.000,A 0.000,B 0.000,C 0.000}
; --------------------------
; ---- Setting tool (TCP) ----
; TOOL_DATA[1] = {FRAME: X 0.000,Y 0.000,Z 10.000,A 0.000,B 0.000,C 0.000}
$TOOL = {FRAME: X 0.000,Y 0.000,Z 10.000,A 0.000,B 0.000,C 0.000}
; $TOOL = TOOL_DATA[1]
; --------------------------
PTP {A1 -90.00780,A2 -59.45620,A3 114.13700,A4 29.35180,A5 -60.28500,A6 -13.70340}
; ---- Setting reference (Base) ----
$BASE = {FRAME: X 0.000,Y 0.000,Z 0.000,A 0.000,B 0.000,C 0.000}
; --------------------------
; ---- Setting tool (TCP) ----
; TOOL_DATA[1] = {FRAME: X 0.000,Y 0.000,Z 10.000,A 0.000,B 0.000,C 0.000}
$TOOL = {FRAME: X 0.000,Y 0.000,Z 10.000,A 0.000,B 0.000,C 0.000}
; $TOOL = TOOL_DATA[1]
; --------------------------
PTP {A1 -95.15830,A2 -59.76330,A3 115.27600,A4 -11.59600,A5 -59.11370,A6 7.99064}
; ---- Setting reference (Base) ----
$BASE = {FRAME: X 0.000,Y 0.000,Z 0.000,A 0.000,B 0.000,C 0.000}
; --------------------------
; ---- Setting tool (TCP) ----
; TOOL_DATA[1] = {FRAME: X 0.000,Y 0.000,Z 10.000,A 0.000,B 0.000,C 0.000}
$TOOL = {FRAME: X 0.000,Y 0.000,Z 10.000,A 0.000,B 0.000,C 0.000}
; $TOOL = TOOL_DATA[1]
; --------------------------
PTP {A1 -95.15830,A2 -59.76330,A3 115.27600,A4 -11.59600,A5 -59.11370,A6 -22.00940}
; ---- Setting reference (Base) ----
$BASE = {FRAME: X 0.000,Y 0.000,Z 0.000,A 0.000,B 0.000,C 0.000}
; --------------------------
; ---- Setting tool (TCP) ----
; TOOL_DATA[1] = {FRAME: X 0.000,Y 0.000,Z 10.000,A 0.000,B 0.000,C 0.000}
$TOOL = {FRAME: X 0.000,Y 0.000,Z 10.000,A 0.000,B 0.000,C 0.000}
; $TOOL = TOOL_DATA[1]
; --------------------------
PTP {A1 -95.15830,A2 -59.76330,A3 115.27600,A4 -11.59600,A5 -59.11370,A6 37.99060}
; ---- Setting reference (Base) ----
$BASE = {FRAME: X 0.000,Y 0.000,Z 0.000,A 0.000,B 0.000,C 0.000}
; --------------------------
; ---- Setting tool (TCP) ----
; TOOL_DATA[1] = {FRAME: X 0.000,Y 0.000,Z 10.000,A 0.000,B 0.000,C 0.000}
$TOOL = {FRAME: X 0.000,Y 0.000,Z 10.000,A 0.000,B 0.000,C 0.000}
; $TOOL = TOOL_DATA[1]
; --------------------------
PTP {A1 -95.15830,A2 -59.76330,A3 115.27600,A4 -11.59600,A5 -59.11370,A6 7.99064}
; ---- Setting reference (Base) ----
$BASE = {FRAME: X 0.000,Y 0.000,Z 0.000,A 0.000,B 0.000,C 0.000}
; --------------------------
; ---- Setting tool (TCP) ----
; TOOL_DATA[1] = {FRAME: X 0.000,Y 0.000,Z 10.000,A 0.000,B 0.000,C 0.000}
$TOOL = {FRAME: X 0.000,Y 0.000,Z 10.000,A 0.000,B 0.000,C 0.000}
; $TOOL = TOOL_DATA[1]
; --------------------------
PTP {A1 -96.33760,A2 -59.53820,A3 114.91300,A4 -12.97570,A5 -59.12120,A6 8.78641}
; ---- Setting reference (Base) ----
$BASE = {FRAME: X 0.000,Y 0.000,Z 0.000,A 0.000,B 0.000,C 0.000}
; --------------------------
; ---- Setting tool (TCP) ----
; TOOL_DATA[1] = {FRAME: X 0.000,Y 0.000,Z 10.000,A 0.000,B 0.000,C 0.000}
$TOOL = {FRAME: X 0.000,Y 0.000,Z 10.000,A 0.000,B 0.000,C 0.000}
; $TOOL = TOOL_DATA[1]
; --------------------------
PTP {A1 -100.82200,A2 -57.37430,A3 110.76800,A4 -50.19480,A5 -68.33370,A6 27.05030}
; ---- Setting reference (Base) ----
$BASE = {FRAME: X 0.000,Y 0.000,Z 0.000,A 0.000,B 0.000,C 0.000}
; --------------------------
; ---- Setting tool (TCP) ----
; TOOL_DATA[1] = {FRAME: X 0.000,Y 0.000,Z 10.000,A 0.000,B 0.000,C 0.000}
$TOOL = {FRAME: X 0.000,Y 0.000,Z 10.000,A 0.000,B 0.000,C 0.000}
; $TOOL = TOOL_DATA[1]
; --------------------------
PTP {A1 -91.18910,A2 -59.31950,A3 113.94900,A4 28.05760,A5 -59.91170,A6 -13.04040}
; ---- Setting reference (Base) ----
$BASE = {FRAME: X 0.000,Y 0.000,Z 0.000,A 0.000,B 0.000,C 0.000}
; --------------------------
; ---- Setting tool (TCP) ----
; TOOL_DATA[1] = {FRAME: X 0.000,Y 0.000,Z 10.000,A 0.000,B 0.000,C 0.000}
$TOOL = {FRAME: X 0.000,Y 0.000,Z 10.000,A 0.000,B 0.000,C 0.000}
; $TOOL = TOOL_DATA[1]
; --------------------------
PTP {A1 -96.33760,A2 -59.53820,A3 114.91300,A4 -12.97570,A5 -59.12120,A6 8.78641}
; ---- Setting reference (Base) ----
$BASE = {FRAME: X 0.000,Y 0.000,Z 0.000,A 0.000,B 0.000,C 0.000}
; --------------------------
; ---- Setting tool (TCP) ----
; TOOL_DATA[1] = {FRAME: X 0.000,Y 0.000,Z 10.000,A 0.000,B 0.000,C 0.000}
$TOOL = {FRAME: X 0.000,Y 0.000,Z 10.000,A 0.000,B 0.000,C 0.000}
; $TOOL = TOOL_DATA[1]
; --------------------------
PTP {A1 -96.33760,A2 -59.53820,A3 114.91300,A4 -12.97570,A5 -59.12120,A6 -21.21360}
; ---- Setting reference (Base) ----
$BASE = {FRAME: X 0.000,Y 0.000,Z 0.000,A 0.000,B 0.000,C 0.000}
; --------------------------
; ---- Setting tool (TCP) ----
; TOOL_DATA[1] = {FRAME: X 0.000,Y 0.000,Z 10.000,A 0.000,B 0.000,C 0.000}
$TOOL = {FRAME: X 0.000,Y 0.000,Z 10.000,A 0.000,B 0.000,C 0.000}
; $TOOL = TOOL_DATA[1]
; --------------------------
PTP {A1 -96.33760,A2 -59.53820,A3 114.91300,A4 -12.97570,A5 -59.12120,A6 38.78640}
; ---- Setting reference (Base) ----
$BASE = {FRAME: X 0.000,Y 0.000,Z 0.000,A 0.000,B 0.000,C 0.000}
; --------------------------
; ---- Setting tool (TCP) ----
; TOOL_DATA[1] = {FRAME: X 0.000,Y 0.000,Z 10.000,A 0.000,B 0.000,C 0.000}
$TOOL = {FRAME: X 0.000,Y 0.000,Z 10.000,A 0.000,B 0.000,C 0.000}
; $TOOL = TOOL_DATA[1]
; --------------------------
PTP {A1 -96.33760,A2 -59.53820,A3 114.91300,A4 -12.97570,A5 -59.12120,A6 8.78641}
; ---- Setting reference (Base) ----
$BASE = {FRAME: X 0.000,Y 0.000,Z 0.000,A 0.000,B 0.000,C 0.000}
; --------------------------
; ---- Setting tool (TCP) ----
; TOOL_DATA[1] = {FRAME: X 0.000,Y 0.000,Z 10.000,A 0.000,B 0.000,C 0.000}
$TOOL = {FRAME: X 0.000,Y 0.000,Z 10.000,A 0.000,B 0.000,C 0.000}
; $TOOL = TOOL_DATA[1]
; --------------------------
PTP {A1 -85.46480,A2 -59.09960,A3 116.62000,A4 -0.29129,A5 -60.55230,A6 1.60269}
; ---- Setting reference (Base) ----
$BASE = {FRAME: X 0.000,Y 0.000,Z 0.000,A 0.000,B 0.000,C 0.000}
; --------------------------
; ---- Setting tool (TCP) ----
; TOOL_DATA[1] = {FRAME: X 0.000,Y 0.000,Z 10.000,A 0.000,B 0.000,C 0.000}
$TOOL = {FRAME: X 0.000,Y 0.000,Z 10.000,A 0.000,B 0.000,C 0.000}
; $TOOL = TOOL_DATA[1]
; --------------------------
PTP {A1 -90.44530,A2 -57.74490,A3 113.99000,A4 -39.07970,A5 -66.15570,A6 20.27550}
; ---- Setting reference (Base) ----
$BASE = {FRAME: X 0.000,Y 0.000,Z 0.000,A 0.000,B 0.000,C 0.000}
; --------------------------
; ---- Setting tool (TCP) ----
; TOOL_DATA[1] = {FRAME: X 0.000,Y 0.000,Z 10.000,A 0.000,B 0.000,C 0.000}
$TOOL = {FRAME: X 0.000,Y 0.000,Z 10.000,A 0.000,B 0.000,C 0.000}
; $TOOL = TOOL_DATA[1]
; --------------------------
PTP {A1 -80.46760,A2 -58.13460,A3 114.08400,A4 39.18140,A5 -64.38710,A6 -17.96040}
; ---- Setting reference (Base) ----
$BASE = {FRAME: X 0.000,Y 0.000,Z 0.000,A 0.000,B 0.000,C 0.000}
; --------------------------
; ---- Setting tool (TCP) ----
; TOOL_DATA[1] = {FRAME: X 0.000,Y 0.000,Z 10.000,A 0.000,B 0.000,C 0.000}
$TOOL = {FRAME: X 0.000,Y 0.000,Z 10.000,A 0.000,B 0.000,C 0.000}
; $TOOL = TOOL_DATA[1]
; --------------------------
PTP {A1 -85.46480,A2 -59.09960,A3 116.62000,A4 -0.29129,A5 -60.55230,A6 1.60269}
; ---- Setting reference (Base) ----
$BASE = {FRAME: X 0.000,Y 0.000,Z 0.000,A 0.000,B 0.000,C 0.000}
; --------------------------
; ---- Setting tool (TCP) ----
; TOOL_DATA[1] = {FRAME: X 0.000,Y 0.000,Z 10.000,A 0.000,B 0.000,C 0.000}
$TOOL = {FRAME: X 0.000,Y 0.000,Z 10.000,A 0.000,B 0.000,C 0.000}
; $TOOL = TOOL_DATA[1]
; --------------------------
PTP {A1 -85.46480,A2 -59.09960,A3 116.62000,A4 -0.29129,A5 -60.55230,A6 -28.39730}
; ---- Setting reference (Base) ----
$BASE = {FRAME: X 0.000,Y 0.000,Z 0.000,A 0.000,B 0.000,C 0.000}
; --------------------------
; ---- Setting tool (TCP) ----
; TOOL_DATA[1] = {FRAME: X 0.000,Y 0.000,Z 10.000,A 0.000,B 0.000,C 0.000}
$TOOL = {FRAME: X 0.000,Y 0.000,Z 10.000,A 0.000,B 0.000,C 0.000}
; $TOOL = TOOL_DATA[1]
; --------------------------
PTP {A1 -85.46480,A2 -59.09960,A3 116.62000,A4 -0.29129,A5 -60.55230,A6 31.60270}
; ---- Setting reference (Base) ----
$BASE = {FRAME: X 0.000,Y 0.000,Z 0.000,A 0.000,B 0.000,C 0.000}
; --------------------------
; ---- Setting tool (TCP) ----
; TOOL_DATA[1] = {FRAME: X 0.000,Y 0.000,Z 10.000,A 0.000,B 0.000,C 0.000}
$TOOL = {FRAME: X 0.000,Y 0.000,Z 10.000,A 0.000,B 0.000,C 0.000}
; $TOOL = TOOL_DATA[1]
; --------------------------
PTP {A1 -85.46480,A2 -59.09960,A3 116.62000,A4 -0.29129,A5 -60.55230,A6 1.60269}
; ---- Setting reference (Base) ----
$BASE = {FRAME: X 0.000,Y 0.000,Z 0.000,A 0.000,B 0.000,C 0.000}
; --------------------------
; ---- Setting tool (TCP) ----
; TOOL_DATA[1] = {FRAME: X 0.000,Y 0.000,Z 10.000,A 0.000,B 0.000,C 0.000}
$TOOL = {FRAME: X 0.000,Y 0.000,Z 10.000,A 0.000,B 0.000,C 0.000}
; $TOOL = TOOL_DATA[1]
; --------------------------
PTP {A1 -86.68380,A2 -59.04150,A3 116.58800,A4 -1.68862,A5 -60.58950,A6 2.35338}
; ---- Setting reference (Base) ----
$BASE = {FRAME: X 0.000,Y 0.000,Z 0.000,A 0.000,B 0.000,C 0.000}
; --------------------------
; ---- Setting tool (TCP) ----
; TOOL_DATA[1] = {FRAME: X 0.000,Y 0.000,Z 10.000,A 0.000,B 0.000,C 0.000}
$TOOL = {FRAME: X 0.000,Y 0.000,Z 10.000,A 0.000,B 0.000,C 0.000}
; $TOOL = TOOL_DATA[1]
; --------------------------
PTP {A1 -91.62360,A2 -57.60460,A3 113.78500,A4 -40.29790,A5 -66.52450,A6 20.87100}
; ---- Setting reference (Base) ----
$BASE = {FRAME: X 0.000,Y 0.000,Z 0.000,A 0.000,B 0.000,C 0.000}
; --------------------------
; ---- Setting tool (TCP) ----
; TOOL_DATA[1] = {FRAME: X 0.000,Y 0.000,Z 10.000,A 0.000,B 0.000,C 0.000}
$TOOL = {FRAME: X 0.000,Y 0.000,Z 10.000,A 0.000,B 0.000,C 0.000}
; $TOOL = TOOL_DATA[1]
; --------------------------
PTP {A1 -81.65240,A2 -58.16300,A3 114.22600,A4 37.91490,A5 -64.06270,A6 -17.30680}
; ---- Setting reference (Base) ----
$BASE = {FRAME: X 0.000,Y 0.000,Z 0.000,A 0.000,B 0.000,C 0.000}
; --------------------------
; ---- Setting tool (TCP) ----
; TOOL_DATA[1] = {FRAME: X 0.000,Y 0.000,Z 10.000,A 0.000,B 0.000,C 0.000}
$TOOL = {FRAME: X 0.000,Y 0.000,Z 10.000,A 0.000,B 0.000,C 0.000}
; $TOOL = TOOL_DATA[1]
; --------------------------
PTP {A1 -86.68380,A2 -59.04150,A3 116.58800,A4 -1.68862,A5 -60.58950,A6 2.35338}
; ---- Setting reference (Base) ----
$BASE = {FRAME: X 0.000,Y 0.000,Z 0.000,A 0.000,B 0.000,C 0.000}
; --------------------------
; ---- Setting tool (TCP) ----
; TOOL_DATA[1] = {FRAME: X 0.000,Y 0.000,Z 10.000,A 0.000,B 0.000,C 0.000}
$TOOL = {FRAME: X 0.000,Y 0.000,Z 10.000,A 0.000,B 0.000,C 0.000}
; $TOOL = TOOL_DATA[1]
; --------------------------
PTP {A1 -86.68380,A2 -59.04150,A3 116.58800,A4 -1.68862,A5 -60.58950,A6 -27.64660}
; ---- Setting reference (Base) ----
$BASE = {FRAME: X 0.000,Y 0.000,Z 0.000,A 0.000,B 0.000,C 0.000}
; --------------------------
; ---- Setting tool (TCP) ----
; TOOL_DATA[1] = {FRAME: X 0.000,Y 0.000,Z 10.000,A 0.000,B 0.000,C 0.000}
$TOOL = {FRAME: X 0.000,Y 0.000,Z 10.000,A 0.000,B 0.000,C 0.000}
; $TOOL = TOOL_DATA[1]
; --------------------------
PTP {A1 -86.68380,A2 -59.04150,A3 116.58800,A4 -1.68862,A5 -60.58950,A6 32.35340}
; ---- Setting reference (Base) ----
$BASE = {FRAME: X 0.000,Y 0.000,Z 0.000,A 0.000,B 0.000,C 0.000}
; --------------------------
; ---- Setting tool (TCP) ----
; TOOL_DATA[1] = {FRAME: X 0.000,Y 0.000,Z 10.000,A 0.000,B 0.000,C 0.000}
$TOOL = {FRAME: X 0.000,Y 0.000,Z 10.000,A 0.000,B 0.000,C 0.000}
; $TOOL = TOOL_DATA[1]
; --------------------------
PTP {A1 -86.68380,A2 -59.04150,A3 116.58800,A4 -1.68862,A5 -60.58950,A6 2.35338}
; ---- Setting reference (Base) ----
$BASE = {FRAME: X 0.000,Y 0.000,Z 0.000,A 0.000,B 0.000,C 0.000}
; --------------------------
; ---- Setting tool (TCP) ----
; TOOL_DATA[1] = {FRAME: X 0.000,Y 0.000,Z 10.000,A 0.000,B 0.000,C 0.000}
$TOOL = {FRAME: X 0.000,Y 0.000,Z 10.000,A 0.000,B 0.000,C 0.000}
; $TOOL = TOOL_DATA[1]
; --------------------------
PTP {A1 -87.90140,A2 -58.96310,A3 116.51400,A4 -3.08373,A5 -60.62110,A6 3.10240}
; ---- Setting reference (Base) ----
$BASE = {FRAME: X 0.000,Y 0.000,Z 0.000,A 0.000,B 0.000,C 0.000}
; --------------------------
; ---- Setting tool (TCP) ----
; TOOL_DATA[1] = {FRAME: X 0.000,Y 0.000,Z 10.000,A 0.000,B 0.000,C 0.000}
$TOOL = {FRAME: X 0.000,Y 0.000,Z 10.000,A 0.000,B 0.000,C 0.000}
; $TOOL = TOOL_DATA[1]
; --------------------------
